QRS_NEXT_CUT()
PTP {E1 29337.004,E2 29337.004}
PTP {X 0,Y 607.899,A -85,B 0,C 180,E1 29337.004,E2 29337.004,E3 0,E4 0,E5 0,E6 0}
QRS_SPEED_INIT()
LIN {X 0,Y 607.899,Z 862.5,A -85,B 0,C 180,E1 29337.004,E2 29337.004,E3 0,E4 0,E5 0,E6 0} C_VEL
LIN {X 0,Y 607.899,Z 754.418,A -85,B 0,C 180,E1 29337.004,E2 29337.004} C_VEL
LIN {X 0,Y 607.899,Z 746.5,A -85,B 0,C 180,E1 29337.004,E2 29337.004} C_VEL
LIN {X 0,Y 607.901,Z 744.678,A -85,B 0,C 180,E1 29336.738,E2 29336.738} C_VEL
LIN {X 0,Y 607.905,Z 753.292,A -85,B 0,C 180,E1 29334.811,E2 29334.811} C_VEL
LIN {X 0,Y 607.912,Z 760.307,A -85,B 0,C 180,E1 29332.821,E2 29332.821} C_VEL
LIN {X 0,Y 607.912,Z 766.021,A -85,B 0,C 180,E1 29330.697,E2 29330.697} C_VEL
LIN {X 0,Y 607.897,Z 769.752,A -85,B 0,C 180,E1 29328.714,E2 29328.714} C_VEL
LIN {X 0,Y 607.897,Z 771.855,A -85,B 0,C 180,E1 29326.689,E2 29326.689} C_VEL
LIN {X 0,Y 607.9,Z 772.434,A -85,B 0,C 180,E1 29324.646,E2 29324.646} C_VEL
LIN {X 0,Y 607.91,Z 771.473,A -85,B 0,C 180,E1 29322.682,E2 29322.682} C_VEL
LIN {X 0,Y 607.91,Z 768.915,A -85,B 0,C 180,E1 29320.697,E2 29320.697} C_VEL
LIN {X 0,Y 607.9,Z 764.827,A -85,B 0,C 180,E1 29318.687,E2 29318.687} C_VEL
LIN {X 0,Y 607.898,Z 759.231,A -85,B 0,C 180,E1 29316.752,E2 29316.752} C_VEL
LIN {X 0,Y 607.902,Z 751.53,A -85,B 0,C 180,E1 29314.684,E2 29314.684} C_VEL
LIN {X 0,Y 607.918,Z 742.857,A -85,B 0,C 180,E1 29312.793,E2 29312.793} C_VEL
LIN {X 0,Y 607.917,Z 732.736,A -85,B 0,C 180,E1 29310.977,E2 29310.977} C_VEL
LIN {X 0,Y 607.91,Z 720.694,A -85,B 0,C 180,E1 29309.128,E2 29309.128} C_VEL
LIN {X 0,Y 607.913,Z 707.235,A -85,B 0,C 180,E1 29307.355,E2 29307.355} C_VEL
LIN {X 0,Y 607.916,Z 692.141,A -85,B 0,C 180,E1 29305.655,E2 29305.655} C_VEL
LIN {X 0,Y 607.915,Z 676.239,A -85,B 0,C 180,E1 29304.104,E2 29304.104} C_VEL
LIN {X 0,Y 607.912,Z 658.424,A -85,B 0,C 180,E1 29302.6,E2 29302.6} C_VEL
LIN {X 0,Y 607.917,Z 640.204,A -85,B 0,C 180,E1 29301.273,E2 29301.273} C_VEL
LIN {X 0,Y 607.917,Z 621.242,A -85,B 0,C 180,E1 29300.103,E2 29300.103} C_VEL
LIN {X 0,Y 607.914,Z 601.356,A -85,B 0,C 180,E1 29299.067,E2 29299.067} C_VEL
LIN {X 0,Y 607.915,Z 581.383,A -85,B 0,C 180,E1 29298.2,E2 29298.2} C_VEL
LIN {X 0,Y 607.915,Z 561.009,A -85,B 0,C 180,E1 29297.504,E2 29297.504} C_VEL
LIN {X 0,Y 607.899,Z 539.165,A -85,B 0,C 180,E1 29296.934,E2 29296.934} C_VEL
LIN {X 0,Y 607.904,Z 518.887,A -85,B 0,C 180,E1 29296.57,E2 29296.57} C_VEL
LIN {X 0,Y 607.912,Z 289.818,A -85,B 0,C 180,E1 29293.507,E2 29293.507} C_VEL
LIN {X 0,Y 607.887,Z 237.014,A -85,B 0,C 180,E1 29292.776,E2 29292.776} C_VEL
LIN {X 0,Y 607.91,Z 237.007,A -85,B 0,C 180,E1 29289.655,E2 29289.655} C_VEL
LIN {X 0,Y 607.874,Z 237.01,A -85,B 0,C 180,E1 29286.459,E2 29286.459} C_VEL
LIN {X 0,Y 607.915,Z 237.008,A -85,B 0,C 180,E1 29283.435,E2 29283.435} C_VEL
LIN {X 0,Y 607.87,Z 237.011,A -85,B 0,C 180,E1 29280.288,E2 29280.288} C_VEL
LIN {X 0,Y 607.913,Z 237.011,A -85,B 0,C 180,E1 29277.157,E2 29277.157} C_VEL
LIN {X 0,Y 607.868,Z 237.01,A -85,B 0,C 180,E1 29274.075,E2 29274.075} C_VEL
LIN {X 0,Y 607.917,Z 237.014,A -85,B 0,C 180,E1 29270.907,E2 29270.907} C_VEL
LIN {X 0,Y 607.874,Z 237.009,A -85,B 0,C 180,E1 29267.764,E2 29267.764} C_VEL
LIN {X 0,Y 607.886,Z 237.013,A -85,B 0,C 180,E1 29264.479,E2 29264.479} C_VEL
LIN {X 0,Y 607.895,Z 237.008,A -85,B 0,C 180,E1 29261.384,E2 29261.384} C_VEL
LIN {X 0,Y 607.872,Z 237.012,A -85,B 0,C 180,E1 29258.228,E2 29258.228} C_VEL
LIN {X 0,Y 607.903,Z 237.008,A -85,B 0,C 180,E1 29255.191,E2 29255.191} C_VEL
LIN {X 0,Y 607.863,Z 237.012,A -85,B 0,C 180,E1 29251.98,E2 29251.98} C_VEL
LIN {X 0,Y 607.917,Z 237.009,A -85,B 0,C 180,E1 29248.87,E2 29248.87} C_VEL
LIN {X 0,Y 607.858,Z 237.011,A -85,B 0,C 180,E1 29245.756,E2 29245.756} C_VEL
LIN {X 0,Y 607.916,Z 237.011,A -85,B 0,C 180,E1 29242.725,E2 29242.725} C_VEL
LIN {X 0,Y 607.856,Z 237.011,A -85,B 0,C 180,E1 29239.672,E2 29239.672} C_VEL
LIN {X 0,Y 607.917,Z 237.012,A -85,B 0,C 180,E1 29236.592,E2 29236.592} C_VEL
LIN {X 0,Y 607.854,Z 237.011,A -85,B 0,C 180,E1 29233.522,E2 29233.522} C_VEL
LIN {X 0,Y 607.918,Z 237.013,A -85,B 0,C 180,E1 29230.456,E2 29230.456} C_VEL
LIN {X 0,Y 607.851,Z 237.012,A -85,B 0,C 180,E1 29227.465,E2 29227.465} C_VEL
LIN {X 0,Y 607.918,Z 237.013,A -85,B 0,C 180,E1 29224.371,E2 29224.371} C_VEL
LIN {X 0,Y 607.849,Z 237.012,A -85,B 0,C 180,E1 29221.403,E2 29221.403} C_VEL
LIN {X 0,Y 607.916,Z 237.012,A -85,B 0,C 180,E1 29218.356,E2 29218.356} C_VEL
LIN {X 0,Y 607.846,Z 237.013,A -85,B 0,C 180,E1 29215.311,E2 29215.311} C_VEL
LIN {X 0,Y 607.919,Z 237.012,A -85,B 0,C 180,E1 29212.279,E2 29212.279} C_VEL
LIN {X 0,Y 607.844,Z 237.013,A -85,B 0,C 180,E1 29209.231,E2 29209.231} C_VEL
LIN {X 0,Y 607.919,Z 237.013,A -85,B 0,C 180,E1 29206.179,E2 29206.179} C_VEL
LIN {X 0,Y 607.84,Z 237.013,A -85,B 0,C 180,E1 29203.177,E2 29203.177} C_VEL
LIN {X 0,Y 607.912,Z 237.013,A -85,B 0,C 180,E1 29200.113,E2 29200.113} C_VEL
LIN {X 0,Y 607.839,Z 237.013,A -85,B 0,C 180,E1 29197.082,E2 29197.082} C_VEL
LIN {X 0,Y 607.915,Z 237.014,A -85,B 0,C 180,E1 29193.999,E2 29193.999} C_VEL
LIN {X 0,Y 607.836,Z 237.014,A -85,B 0,C 180,E1 29190.986,E2 29190.986} C_VEL
LIN {X 0,Y 607.915,Z 237.013,A -85,B 0,C 180,E1 29187.951,E2 29187.951} C_VEL
LIN {X 0,Y 607.834,Z 237.014,A -85,B 0,C 180,E1 29184.903,E2 29184.903} C_VEL
LIN {X 0,Y 607.904,Z 237.014,A -85,B 0,C 180,E1 29181.921,E2 29181.921} C_VEL
LIN {X 0,Y 607.833,Z 237.014,A -85,B 0,C 180,E1 29178.907,E2 29178.907} C_VEL
LIN {X 0,Y 607.888,Z 237.014,A -85,B 0,C 180,E1 29175.941,E2 29175.941} C_VEL
LIN {X 0,Y 607.833,Z 237.015,A -85,B 0,C 180,E1 29172.926,E2 29172.926} C_VEL
LIN {X 0,Y 607.844,Z 237.014,A -85,B 0,C 180,E1 29170.231,E2 29170.231} C_VEL
LIN {X 0,Y 607.839,Z 237.015,A -85,B 0,C 180,E1 29166.99,E2 29166.99} C_VEL
LIN {X 0,Y 607.835,Z 237.015,A -85,B 0,C 180,E1 29164.244,E2 29164.244} C_VEL
LIN {X 0,Y 607.843,Z 237.015,A -85,B 0,C 180,E1 29160.941,E2 29160.941} C_VEL
LIN {X 0,Y 607.834,Z 237.015,A -85,B 0,C 180,E1 29158.208,E2 29158.208} C_VEL
LIN {X 0,Y 607.858,Z 237.014,A -85,B 0,C 180,E1 29154.998,E2 29154.998} C_VEL
LIN {X 0,Y 607.836,Z 237.014,A -85,B 0,C 180,E1 29152.152,E2 29152.152} C_VEL
LIN {X 0,Y 607.871,Z 237.014,A -85,B 0,C 180,E1 29148.999,E2 29148.999} C_VEL
LIN {X 0,Y 607.834,Z 237.014,A -85,B 0,C 180,E1 29146.2,E2 29146.2} C_VEL
LIN {X 0,Y 607.894,Z 237.013,A -85,B 0,C 180,E1 29143.074,E2 29143.074} C_VEL
LIN {X 0,Y 607.835,Z 237.014,A -85,B 0,C 180,E1 29140.192,E2 29140.192} C_VEL
LIN {X 0,Y 607.915,Z 237.013,A -85,B 0,C 180,E1 29137.159,E2 29137.159} C_VEL
LIN {X 0,Y 607.837,Z 237.013,A -85,B 0,C 180,E1 29134.126,E2 29134.126} C_VEL
LIN {X 0,Y 607.914,Z 237.014,A -85,B 0,C 180,E1 29131.082,E2 29131.082} C_VEL
LIN {X 0,Y 607.84,Z 237.013,A -85,B 0,C 180,E1 29128.077,E2 29128.077} C_VEL
LIN {X 0,Y 607.918,Z 237.012,A -85,B 0,C 180,E1 29124.969,E2 29124.969} C_VEL
LIN {X 0,Y 607.843,Z 237.013,A -85,B 0,C 180,E1 29121.913,E2 29121.913} C_VEL
LIN {X 0,Y 607.918,Z 237.012,A -85,B 0,C 180,E1 29118.86,E2 29118.86} C_VEL
LIN {X 0,Y 607.845,Z 237.013,A -85,B 0,C 180,E1 29115.82,E2 29115.82} C_VEL
LIN {X 0,Y 607.918,Z 237.012,A -85,B 0,C 180,E1 29112.785,E2 29112.785} C_VEL
LIN {X 0,Y 607.848,Z 237.012,A -85,B 0,C 180,E1 29109.78,E2 29109.78} C_VEL
LIN {X 0,Y 607.919,Z 237.08,A -85,B 0,C 180,E1 29106.651,E2 29106.651} C_VEL
LIN {X 0,Y 607.92,Z 284.175,A -85,B 0,C 180,E1 29103.546,E2 29103.546} C_VEL
LIN {X 0,Y 607.916,Z 302.922,A -85,B 0,C 180,E1 29102.36,E2 29102.36} C_VEL
LIN {X 0,Y 607.905,Z 524.312,A -85,B 0,C 180,E1 29099.375,E2 29099.375} C_VEL
LIN {X 0,Y 607.903,Z 607.752,A -85,B 0,C 180,E1 29098.246,E2 29098.246} C_VEL
LIN {X 0,Y 607.908,Z 628.255,A -85,B 0,C 180,E1 29097.805,E2 29097.805} C_VEL
LIN {X 0,Y 607.907,Z 648.842,A -85,B 0,C 180,E1 29097.208,E2 29097.208} C_VEL
LIN {X 0,Y 607.913,Z 669.605,A -85,B 0,C 180,E1 29096.416,E2 29096.416} C_VEL
LIN {X 0,Y 607.918,Z 690.768,A -85,B 0,C 180,E1 29095.42,E2 29095.42} C_VEL
LIN {X 0,Y 607.916,Z 710.107,A -85,B 0,C 180,E1 29094.331,E2 29094.331} C_VEL
LIN {X 0,Y 607.914,Z 728.578,A -85,B 0,C 180,E1 29093.094,E2 29093.094} C_VEL
LIN {X 0,Y 607.911,Z 746.777,A -85,B 0,C 180,E1 29091.677,E2 29091.677} C_VEL
LIN {X 0,Y 607.913,Z 763.663,A -85,B 0,C 180,E1 29090.154,E2 29090.154} C_VEL
LIN {X 0,Y 607.918,Z 779.474,A -85,B 0,C 180,E1 29088.506,E2 29088.506} C_VEL
LIN {X 0,Y 607.913,Z 793.414,A -85,B 0,C 180,E1 29086.816,E2 29086.816} C_VEL
LIN {X 0,Y 607.918,Z 805.908,A -85,B 0,C 180,E1 29085.061,E2 29085.061} C_VEL
LIN {X 0,Y 607.919,Z 817.422,A -85,B 0,C 180,E1 29083.176,E2 29083.176} C_VEL
LIN {X 0,Y 607.912,Z 827.065,A -85,B 0,C 180,E1 29081.286,E2 29081.286} C_VEL
LIN {X 0,Y 607.911,Z 835.467,A -85,B 0,C 180,E1 29079.275,E2 29079.275} C_VEL
LIN {X 0,Y 607.91,Z 842.13,A -85,B 0,C 180,E1 29077.275,E2 29077.275} C_VEL
LIN {X 0,Y 607.914,Z 847.016,A -85,B 0,C 180,E1 29075.284,E2 29075.284} C_VEL
LIN {X 0,Y 607.917,Z 850.447,A -85,B 0,C 180,E1 29073.205,E2 29073.205} C_VEL
LIN {X 0,Y 607.91,Z 852.21,A -85,B 0,C 180,E1 29071.224,E2 29071.224} C_VEL
LIN {X 0,Y 607.902,Z 852.328,A -85,B 0,C 180,E1 29069.245,E2 29069.245} C_VEL
LIN {X 0,Y 607.908,Z 850.894,A -85,B 0,C 180,E1 29067.171,E2 29067.171} C_VEL
LIN {X 0,Y 607.912,Z 847.985,A -85,B 0,C 180,E1 29065.187,E2 29065.187} C_VEL
LIN {X 0,Y 607.915,Z 843.396,A -85,B 0,C 180,E1 29063.198,E2 29063.198} C_VEL
LIN {X 0,Y 607.906,Z 837.234,A -85,B 0,C 180,E1 29061.201,E2 29061.201} C_VEL
LIN {X 0,Y 607.899,Z 829.652,A -85,B 0,C 180,E1 29059.288,E2 29059.288} C_VEL
LIN {X 0,Y 607.899,Z 820.322,A -85,B 0,C 180,E1 29057.363,E2 29057.363} C_VEL
LIN {X 0,Y 607.904,Z 809.74,A -85,B 0,C 180,E1 29055.521,E2 29055.521} C_VEL
LIN {X 0,Y 607.911,Z 797.735,A -85,B 0,C 180,E1 29053.763,E2 29053.763} C_VEL
LIN {X 0,Y 607.906,Z 783.709,A -85,B 0,C 180,E1 29051.987,E2 29051.987} C_VEL
LIN {X 0,Y 607.908,Z 768.706,A -85,B 0,C 180,E1 29050.345,E2 29050.345} C_VEL
LIN {X 0,Y 607.916,Z 751.689,A -85,B 0,C 180,E1 29048.735,E2 29048.735} C_VEL
LIN {X 0,Y 607.918,Z 734.236,A -85,B 0,C 180,E1 29047.323,E2 29047.323} C_VEL
LIN {X 0,Y 607.915,Z 715.722,A -85,B 0,C 180,E1 29046.03,E2 29046.03} C_VEL
LIN {X 0,Y 607.918,Z 696.693,A -85,B 0,C 180,E1 29044.89,E2 29044.89} C_VEL
LIN {X 0,Y 607.9,Z 676.895,A -85,B 0,C 180,E1 29043.902,E2 29043.902} C_VEL
LIN {X 0,Y 607.907,Z 656.203,A -85,B 0,C 180,E1 29043.057,E2 29043.057} C_VEL
LIN {X 0,Y 607.918,Z 636.195,A -85,B 0,C 180,E1 29042.402,E2 29042.402} C_VEL
LIN {X 0,Y 607.904,Z 615.922,A -85,B 0,C 180,E1 29041.913,E2 29041.913} C_VEL
LIN {X 0,Y 607.914,Z 594.386,A -85,B 0,C 180,E1 29041.552,E2 29041.552} C_VEL
LIN {X 0,Y 607.881,Z 369.433,A -85,B 0,C 180,E1 29038.545,E2 29038.545} C_VEL
LIN {X 0,Y 607.916,Z 302.484,A -85,B 0,C 180,E1 29037.631,E2 29037.631} C_VEL
LIN {X 0,Y 607.865,Z 256.986,A -85,B 0,C 180,E1 29034.672,E2 29034.672} C_VEL
LIN {X 0,Y 607.919,Z 237.013,A -85,B 0,C 180,E1 29033.342,E2 29033.342} C_VEL
LIN {X 0,Y 607.846,Z 237.013,A -85,B 0,C 180,E1 29030.217,E2 29030.217} C_VEL
LIN {X 0,Y 607.919,Z 237.013,A -85,B 0,C 180,E1 29027.185,E2 29027.185} C_VEL
LIN {X 0,Y 607.843,Z 237.013,A -85,B 0,C 180,E1 29024.177,E2 29024.177} C_VEL
LIN {X 0,Y 607.919,Z 237.013,A -85,B 0,C 180,E1 29021.124,E2 29021.124} C_VEL
LIN {X 0,Y 607.838,Z 237.014,A -85,B 0,C 180,E1 29018.087,E2 29018.087} C_VEL
LIN {X 0,Y 607.919,Z 237.014,A -85,B 0,C 180,E1 29015.008,E2 29015.008} C_VEL
LIN {X 0,Y 607.834,Z 237.014,A -85,B 0,C 180,E1 29011.919,E2 29011.919} C_VEL
LIN {X 0,Y 607.906,Z 237.016,A -85,B 0,C 180,E1 29008.919,E2 29008.919} C_VEL
LIN {X 0,Y 607.829,Z 237.015,A -85,B 0,C 180,E1 29005.949,E2 29005.949} C_VEL
LIN {X 0,Y 607.892,Z 237.015,A -85,B 0,C 180,E1 29003.046,E2 29003.046} C_VEL
LIN {X 0,Y 607.829,Z 237.015,A -85,B 0,C 180,E1 29000.009,E2 29000.009} C_VEL
LIN {X 0,Y 607.869,Z 237.048,A -85,B 0,C 180,E1 28997.124,E2 28997.124} C_VEL
LIN {X 0,Y 607.9,Z 476.426,A -85,B 0,C 180,E1 28993.905,E2 28993.905} C_VEL
LIN {X 0,Y 607.902,Z 529.091,A -85,B 0,C 180,E1 28993.18,E2 28993.18} C_VEL
LIN {X 0,Y 607.918,Z 549.308,A -85,B 0,C 180,E1 28992.733,E2 28992.733} C_VEL
LIN {X 0,Y 607.901,Z 570.449,A -85,B 0,C 180,E1 28992.106,E2 28992.106} C_VEL
LIN {X 0,Y 607.901,Z 590.463,A -85,B 0,C 180,E1 28991.336,E2 28991.336} C_VEL
LIN {X 0,Y 607.919,Z 610.908,A -85,B 0,C 180,E1 28990.368,E2 28990.368} C_VEL
LIN {X 0,Y 607.917,Z 630.263,A -85,B 0,C 180,E1 28989.277,E2 28989.277} C_VEL
LIN {X 0,Y 607.914,Z 648.753,A -85,B 0,C 180,E1 28988.038,E2 28988.038} C_VEL
LIN {X 0,Y 607.913,Z 667.016,A -85,B 0,C 180,E1 28986.612,E2 28986.612} C_VEL
LIN {X 0,Y 607.915,Z 683.795,A -85,B 0,C 180,E1 28985.097,E2 28985.097} C_VEL
LIN {X 0,Y 607.915,Z 699.232,A -85,B 0,C 180,E1 28983.49,E2 28983.49} C_VEL
LIN {X 0,Y 607.916,Z 713.253,A -85,B 0,C 180,E1 28981.792,E2 28981.792} C_VEL
LIN {X 0,Y 607.914,Z 726.007,A -85,B 0,C 180,E1 28980.001,E2 28980.001} C_VEL
LIN {X 0,Y 607.913,Z 737.503,A -85,B 0,C 180,E1 28978.116,E2 28978.116} C_VEL
LIN {X 0,Y 607.901,Z 744.678,A -85,B 0,C 180,E1 28976.738,E2 28976.738} C_VEL
LIN {X 0,Y 606.904,Z 747.955,A -85,B 0,C 180,E1 28976.076,E2 28976.076} C_VEL
LIN {X 0,Y 600.672,Z 755.675,A -85,B 0,C 180,E1 28974.293,E2 28974.293} C_VEL
LIN {X 0,Y 599.922,Z 757.876,A -85,B 0,C 180,E1 28973.696,E2 28973.696} C_VEL
LIN {X 0,Y 599.92,Z 763.885,A -85,B 0,C 180,E1 28971.664,E2 28971.664} C_VEL
LIN {X 0,Y 599.91,Z 768.491,A -85,B 0,C 180,E1 28969.528,E2 28969.528} C_VEL
LIN {X 0,Y 599.902,Z 771.287,A -85,B 0,C 180,E1 28967.488,E2 28967.488} C_VEL
LIN {X 0,Y 599.91,Z 772.4,A -85,B 0,C 180,E1 28965.425,E2 28965.425} C_VEL
LIN {X 0,Y 599.917,Z 771.889,A -85,B 0,C 180,E1 28963.244,E2 28963.244} C_VEL
LIN {X 0,Y 599.915,Z 769.843,A -85,B 0,C 180,E1 28961.204,E2 28961.204} C_VEL
LIN {X 0,Y 599.918,Z 766.178,A -85,B 0,C 180,E1 28959.209,E2 28959.209} C_VEL
LIN {X 0,Y 599.921,Z 760.511,A -85,B 0,C 180,E1 28957.048,E2 28957.048} C_VEL
LIN {X 0,Y 599.933,Z 753.6,A -85,B 0,C 180,E1 28955.046,E2 28955.046} C_VEL
LIN {X 0,Y 599.947,Z 744.835,A -85,B 0,C 180,E1 28953.046,E2 28953.046} C_VEL
LIN {X 0,Y 599.973,Z 733.944,A -85,B 0,C 180,E1 28950.993,E2 28950.993} C_VEL
LIN {X 0,Y 600.007,Z 722.136,A -85,B 0,C 180,E1 28949.116,E2 28949.116} C_VEL
LIN {X 0,Y 600.052,Z 708.647,A -85,B 0,C 180,E1 28947.297,E2 28947.297} C_VEL
LIN {X 0,Y 600.123,Z 693.662,A -85,B 0,C 180,E1 28945.56,E2 28945.56} C_VEL
LIN {X 0,Y 600.203,Z 677.026,A -85,B 0,C 180,E1 28943.896,E2 28943.896} C_VEL
LIN {X 0,Y 600.292,Z 660.221,A -85,B 0,C 180,E1 28942.441,E2 28942.441} C_VEL
LIN {X 0,Y 600.386,Z 641.597,A -85,B 0,C 180,E1 28941.053,E2 28941.053} C_VEL
LIN {X 0,Y 600.481,Z 622.419,A -85,B 0,C 180,E1 28939.843,E2 28939.843} C_VEL
LIN {X 0,Y 600.59,Z 601.315,A -85,B 0,C 180,E1 28938.725,E2 28938.725} C_VEL
LIN {X 0,Y 600.687,Z 580.897,A -85,B 0,C 180,E1 28937.833,E2 28937.833} C_VEL
LIN {X 0,Y 600.755,Z 559.86,A -85,B 0,C 180,E1 28937.113,E2 28937.113} C_VEL
LIN {X 0,Y 600.816,Z 537.813,A -85,B 0,C 180,E1 28936.545,E2 28936.545} C_VEL
LIN {X 0,Y 600.867,Z 516.414,A -85,B 0,C 180,E1 28936.169,E2 28936.169} C_VEL
LIN {X 0,Y 601.082,Z 290.741,A -85,B 0,C 180,E1 28933.121,E2 28933.121} C_VEL
LIN {X 0,Y 600.973,Z 241.06,A -85,B 0,C 180,E1 28932.427,E2 28932.427} C_VEL
LIN {X 0,Y 599.935,Z 238.001,A -85,B 0,C 180,E1 28932.299,E2 28932.299} C_VEL
LIN {X 0,Y 599.976,Z 238.003,A -85,B 0,C 180,E1 28929.169,E2 28929.169} C_VEL
LIN {X 0,Y 599.941,Z 237.996,A -85,B 0,C 180,E1 28926.038,E2 28926.038} C_VEL
LIN {X 0,Y 599.959,Z 238.003,A -85,B 0,C 180,E1 28922.795,E2 28922.795} C_VEL
LIN {X 0,Y 599.973,Z 237.995,A -85,B 0,C 180,E1 28919.556,E2 28919.556} C_VEL
LIN {X 0,Y 599.932,Z 238.001,A -85,B 0,C 180,E1 28916.317,E2 28916.317} C_VEL
LIN {X 0,Y 599.977,Z 237.997,A -85,B 0,C 180,E1 28913.264,E2 28913.264} C_VEL
LIN {X 0,Y 599.93,Z 238,A -85,B 0,C 180,E1 28910.182,E2 28910.182} C_VEL
LIN {X 0,Y 599.975,Z 237.999,A -85,B 0,C 180,E1 28907.057,E2 28907.057} C_VEL
LIN {X 0,Y 599.926,Z 237.999,A -85,B 0,C 180,E1 28903.985,E2 28903.985} C_VEL
LIN {X 0,Y 599.976,Z 238.002,A -85,B 0,C 180,E1 28900.855,E2 28900.855} C_VEL
LIN {X 0,Y 599.925,Z 237.999,A -85,B 0,C 180,E1 28897.759,E2 28897.759} C_VEL
LIN {X 0,Y 599.973,Z 238.003,A -85,B 0,C 180,E1 28894.589,E2 28894.589} C_VEL
LIN {X 0,Y 599.929,Z 237.998,A -85,B 0,C 180,E1 28891.529,E2 28891.529} C_VEL
LIN {X 0,Y 599.945,Z 238.002,A -85,B 0,C 180,E1 28888.282,E2 28888.282} C_VEL
LIN {X 0,Y 599.943,Z 237.997,A -85,B 0,C 180,E1 28885.221,E2 28885.221} C_VEL
LIN {X 0,Y 599.925,Z 238.001,A -85,B 0,C 180,E1 28881.953,E2 28881.953} C_VEL
LIN {X 0,Y 599.969,Z 237.998,A -85,B 0,C 180,E1 28878.855,E2 28878.855} C_VEL
LIN {X 0,Y 599.917,Z 238.001,A -85,B 0,C 180,E1 28875.721,E2 28875.721} C_VEL
LIN {X 0,Y 599.975,Z 237.999,A -85,B 0,C 180,E1 28872.645,E2 28872.645} C_VEL
LIN {X 0,Y 599.913,Z 238.001,A -85,B 0,C 180,E1 28869.514,E2 28869.514} C_VEL
LIN {X 0,Y 599.979,Z 238.001,A -85,B 0,C 180,E1 28866.423,E2 28866.423} C_VEL
LIN {X 0,Y 599.911,Z 238.001,A -85,B 0,C 180,E1 28863.364,E2 28863.364} C_VEL
LIN {X 0,Y 599.978,Z 238.004,A -85,B 0,C 180,E1 28860.225,E2 28860.225} C_VEL
LIN {X 0,Y 599.912,Z 238,A -85,B 0,C 180,E1 28857.136,E2 28857.136} C_VEL
LIN {X 0,Y 599.946,Z 238.003,A -85,B 0,C 180,E1 28853.925,E2 28853.925} C_VEL
LIN {X 0,Y 599.909,Z 238.001,A -85,B 0,C 180,E1 28851.074,E2 28851.074} C_VEL
LIN {X 0,Y 599.947,Z 238.004,A -85,B 0,C 180,E1 28847.867,E2 28847.867} C_VEL
LIN {X 0,Y 599.907,Z 238.001,A -85,B 0,C 180,E1 28844.962,E2 28844.962} C_VEL
LIN {X 0,Y 599.948,Z 238.004,A -85,B 0,C 180,E1 28841.805,E2 28841.805} C_VEL
LIN {X 0,Y 599.904,Z 238.002,A -85,B 0,C 180,E1 28838.893,E2 28838.893} C_VEL
LIN {X 0,Y 599.949,Z 238.003,A -85,B 0,C 180,E1 28835.748,E2 28835.748} C_VEL
LIN {X 0,Y 599.901,Z 238.002,A -85,B 0,C 180,E1 28832.796,E2 28832.796} C_VEL
LIN {X 0,Y 599.947,Z 238.004,A -85,B 0,C 180,E1 28829.666,E2 28829.666} C_VEL
LIN {X 0,Y 599.898,Z 238.002,A -85,B 0,C 180,E1 28826.742,E2 28826.742} C_VEL
LIN {X 0,Y 599.959,Z 238.004,A -85,B 0,C 180,E1 28823.679,E2 28823.679} C_VEL
LIN {X 0,Y 599.894,Z 238.003,A -85,B 0,C 180,E1 28820.69,E2 28820.69} C_VEL
LIN {X 0,Y 599.957,Z 238.004,A -85,B 0,C 180,E1 28817.591,E2 28817.591} C_VEL
LIN {X 0,Y 599.891,Z 238.003,A -85,B 0,C 180,E1 28814.674,E2 28814.674} C_VEL
LIN {X 0,Y 599.972,Z 238.004,A -85,B 0,C 180,E1 28811.632,E2 28811.632} C_VEL
LIN {X 0,Y 599.889,Z 238.004,A -85,B 0,C 180,E1 28808.626,E2 28808.626} C_VEL
LIN {X 0,Y 599.967,Z 238.004,A -85,B 0,C 180,E1 28805.641,E2 28805.641} C_VEL
LIN {X 0,Y 599.886,Z 238.004,A -85,B 0,C 180,E1 28802.578,E2 28802.578} C_VEL
LIN {X 0,Y 599.961,Z 238.004,A -85,B 0,C 180,E1 28799.617,E2 28799.617} C_VEL
LIN {X 0,Y 599.891,Z 238.004,A -85,B 0,C 180,E1 28796.559,E2 28796.559} C_VEL
LIN {X 0,Y 599.956,Z 238.003,A -85,B 0,C 180,E1 28793.588,E2 28793.588} C_VEL
LIN {X 0,Y 599.893,Z 238.003,A -85,B 0,C 180,E1 28790.501,E2 28790.501} C_VEL
LIN {X 0,Y 599.947,Z 238.004,A -85,B 0,C 180,E1 28787.577,E2 28787.577} C_VEL
LIN {X 0,Y 599.897,Z 238.003,A -85,B 0,C 180,E1 28784.433,E2 28784.433} C_VEL
LIN {X 0,Y 599.948,Z 238.004,A -85,B 0,C 180,E1 28781.487,E2 28781.487} C_VEL
LIN {X 0,Y 599.9,Z 238.002,A -85,B 0,C 180,E1 28778.386,E2 28778.386} C_VEL
LIN {X 0,Y 599.942,Z 238.003,A -85,B 0,C 180,E1 28775.481,E2 28775.481} C_VEL
LIN {X 0,Y 599.907,Z 238.002,A -85,B 0,C 180,E1 28772.396,E2 28772.396} C_VEL
LIN {X 0,Y 599.931,Z 238.003,A -85,B 0,C 180,E1 28769.498,E2 28769.498} C_VEL
LIN {X 0,Y 599.908,Z 238.002,A -85,B 0,C 180,E1 28766.268,E2 28766.268} C_VEL
LIN {X 0,Y 599.939,Z 238.004,A -85,B 0,C 180,E1 28763.37,E2 28763.37} C_VEL
LIN {X 0,Y 599.911,Z 238.002,A -85,B 0,C 180,E1 28760.202,E2 28760.202} C_VEL
LIN {X 0,Y 599.941,Z 238.004,A -85,B 0,C 180,E1 28757.288,E2 28757.288} C_VEL
LIN {X 0,Y 599.912,Z 238.002,A -85,B 0,C 180,E1 28754.082,E2 28754.082} C_VEL
LIN {X 0,Y 599.965,Z 238.004,A -85,B 0,C 180,E1 28751.04,E2 28751.04} C_VEL
LIN {X 0,Y 599.913,Z 238.003,A -85,B 0,C 180,E1 28747.95,E2 28747.95} C_VEL
LIN {X 0,Y 599.978,Z 238.232,A -85,B 0,C 180,E1 28747.139,E2 28747.139} C_VEL
LIN {X 0,Y 601.065,Z 241.208,A -85,B 0,C 180,E1 28746.857,E2 28746.857} C_VEL
LIN {X 0,Y 600.904,Z 286.795,A -85,B 0,C 180,E1 28743.818,E2 28743.818} C_VEL
LIN {X 0,Y 600.96,Z 303.158,A -85,B 0,C 180,E1 28742.778,E2 28742.778} C_VEL
LIN {X 0,Y 600.982,Z 464.512,A -85,B 0,C 180,E1 28740.557,E2 28740.557} C_VEL
LIN {X 0,Y 600.847,Z 607.966,A -85,B 0,C 180,E1 28738.605,E2 28738.605} C_VEL
LIN {X 0,Y 600.789,Z 628.958,A -85,B 0,C 180,E1 28738.145,E2 28738.145} C_VEL
LIN {X 0,Y 600.712,Z 649.582,A -85,B 0,C 180,E1 28737.534,E2 28737.534} C_VEL
LIN {X 0,Y 600.646,Z 669.608,A -85,B 0,C 180,E1 28736.761,E2 28736.761} C_VEL
LIN {X 0,Y 600.54,Z 690.771,A -85,B 0,C 180,E1 28735.755,E2 28735.755} C_VEL
LIN {X 0,Y 600.445,Z 710.128,A -85,B 0,C 180,E1 28734.652,E2 28734.652} C_VEL
LIN {X 0,Y 600.355,Z 728.425,A -85,B 0,C 180,E1 28733.414,E2 28733.414} C_VEL
LIN {X 0,Y 600.25,Z 746.287,A -85,B 0,C 180,E1 28732.01,E2 28732.01} C_VEL
LIN {X 0,Y 600.165,Z 763.156,A -85,B 0,C 180,E1 28730.477,E2 28730.477} C_VEL
LIN {X 0,Y 600.102,Z 778.669,A -85,B 0,C 180,E1 28728.85,E2 28728.85} C_VEL
LIN {X 0,Y 600.048,Z 792.568,A -85,B 0,C 180,E1 28727.152,E2 28727.152} C_VEL
LIN {X 0,Y 599.999,Z 805.91,A -85,B 0,C 180,E1 28725.265,E2 28725.265} C_VEL
LIN {X 0,Y 599.958,Z 817.217,A -85,B 0,C 180,E1 28723.393,E2 28723.393} C_VEL
LIN {X 0,Y 599.931,Z 826.837,A -85,B 0,C 180,E1 28721.486,E2 28721.486} C_VEL
LIN {X 0,Y 599.915,Z 835.113,A -85,B 0,C 180,E1 28719.496,E2 28719.496} C_VEL
LIN {X 0,Y 599.912,Z 841.875,A -85,B 0,C 180,E1 28717.469,E2 28717.469} C_VEL
LIN {X 0,Y 599.915,Z 846.811,A -85,B 0,C 180,E1 28715.45,E2 28715.45} C_VEL
LIN {X 0,Y 599.916,Z 850.37,A -85,B 0,C 180,E1 28713.313,E2 28713.313} C_VEL
LIN {X 0,Y 599.909,Z 852.21,A -85,B 0,C 180,E1 28711.241,E2 28711.241} C_VEL
LIN {X 0,Y 599.902,Z 852.328,A -85,B 0,C 180,E1 28709.235,E2 28709.235} C_VEL
LIN {X 0,Y 599.909,Z 850.894,A -85,B 0,C 180,E1 28707.133,E2 28707.133} C_VEL
LIN {X 0,Y 599.914,Z 847.985,A -85,B 0,C 180,E1 28705.123,E2 28705.123} C_VEL
LIN {X 0,Y 599.92,Z 843.396,A -85,B 0,C 180,E1 28703.107,E2 28703.107} C_VEL
LIN {X 0,Y 599.924,Z 837.235,A -85,B 0,C 180,E1 28701.083,E2 28701.083} C_VEL
LIN {X 0,Y 599.923,Z 829.653,A -85,B 0,C 180,E1 28699.144,E2 28699.144} C_VEL
LIN {X 0,Y 599.942,Z 820.093,A -85,B 0,C 180,E1 28697.15,E2 28697.15} C_VEL
LIN {X 0,Y 599.978,Z 809.104,A -85,B 0,C 180,E1 28695.227,E2 28695.227} C_VEL
LIN {X 0,Y 600.013,Z 797.029,A -85,B 0,C 180,E1 28693.443,E2 28693.443} C_VEL
LIN {X 0,Y 600.082,Z 782.859,A -85,B 0,C 180,E1 28691.644,E2 28691.644} C_VEL
LIN {X 0,Y 600.156,Z 767.187,A -85,B 0,C 180,E1 28689.928,E2 28689.928} C_VEL
LIN {X 0,Y 600.243,Z 750.582,A -85,B 0,C 180,E1 28688.356,E2 28688.356} C_VEL
LIN {X 0,Y 600.318,Z 732.788,A -85,B 0,C 180,E1 28686.906,E2 28686.906} C_VEL
LIN {X 0,Y 600.421,Z 714.12,A -85,B 0,C 180,E1 28685.607,E2 28685.607} C_VEL
LIN {X 0,Y 600.533,Z 693.714,A -85,B 0,C 180,E1 28684.401,E2 28684.401} C_VEL
LIN {X 0,Y 600.607,Z 674.531,A -85,B 0,C 180,E1 28683.449,E2 28683.449} C_VEL
LIN {X 0,Y 600.695,Z 653.94,A -85,B 0,C 180,E1 28682.624,E2 28682.624} C_VEL
LIN {X 0,Y 600.79,Z 632.305,A -85,B 0,C 180,E1 28681.942,E2 28681.942} C_VEL
LIN {X 0,Y 600.828,Z 612.544,A -85,B 0,C 180,E1 28681.482,E2 28681.482} C_VEL
LIN {X 0,Y 600.891,Z 583.533,A -85,B 0,C 180,E1 28681.043,E2 28681.043} C_VEL
LIN {X 0,Y 601.06,Z 360.357,A -85,B 0,C 180,E1 28678.021,E2 28678.021} C_VEL
LIN {X 0,Y 600.94,Z 303.057,A -85,B 0,C 180,E1 28677.22,E2 28677.22} C_VEL
LIN {X 0,Y 600.956,Z 260.62,A -85,B 0,C 180,E1 28674.448,E2 28674.448} C_VEL
LIN {X 0,Y 601.064,Z 241.21,A -85,B 0,C 180,E1 28673.143,E2 28673.143} C_VEL
LIN {X 0,Y 599.94,Z 238.006,A -85,B 0,C 180,E1 28672.81,E2 28672.81} C_VEL
LIN {X 0,Y 599.916,Z 238.002,A -85,B 0,C 180,E1 28669.907,E2 28669.907} C_VEL
LIN {X 0,Y 599.924,Z 238.004,A -85,B 0,C 180,E1 28666.607,E2 28666.607} C_VEL
LIN {X 0,Y 599.917,Z 238.002,A -85,B 0,C 180,E1 28663.762,E2 28663.762} C_VEL
LIN {X 0,Y 599.911,Z 238.003,A -85,B 0,C 180,E1 28660.417,E2 28660.417} C_VEL
LIN {X 0,Y 599.92,Z 238.002,A -85,B 0,C 180,E1 28657.59,E2 28657.59} C_VEL
LIN {X 0,Y 599.912,Z 238.004,A -85,B 0,C 180,E1 28654.403,E2 28654.403} C_VEL
LIN {X 0,Y 599.912,Z 238.003,A -85,B 0,C 180,E1 28651.557,E2 28651.557} C_VEL
LIN {X 0,Y 599.902,Z 238.004,A -85,B 0,C 180,E1 28648.252,E2 28648.252} C_VEL
LIN {X 0,Y 599.907,Z 238.004,A -85,B 0,C 180,E1 28645.469,E2 28645.469} C_VEL
LIN {X 0,Y 599.901,Z 238.005,A -85,B 0,C 180,E1 28642.232,E2 28642.232} C_VEL
LIN {X 0,Y 599.898,Z 238.005,A -85,B 0,C 180,E1 28639.473,E2 28639.473} C_VEL
LIN {X 0,Y 599.912,Z 238.159,A -85,B 0,C 180,E1 28637.588,E2 28637.588} C_VEL
LIN {X 0,Y 601.095,Z 242.026,A -85,B 0,C 180,E1 28637.462,E2 28637.462} C_VEL
LIN {X 0,Y 600.895,Z 479.792,A -85,B 0,C 180,E1 28634.23,E2 28634.23} C_VEL
LIN {X 0,Y 600.837,Z 529.695,A -85,B 0,C 180,E1 28633.531,E2 28633.531} C_VEL
LIN {X 0,Y 600.797,Z 550.734,A -85,B 0,C 180,E1 28633.055,E2 28633.055} C_VEL
LIN {X 0,Y 600.694,Z 572.744,A -85,B 0,C 180,E1 28632.376,E2 28632.376} C_VEL
LIN {X 0,Y 600.619,Z 593.04,A -85,B 0,C 180,E1 28631.573,E2 28631.573} C_VEL
LIN {X 0,Y 600.537,Z 612.809,A -85,B 0,C 180,E1 28630.602,E2 28630.602} C_VEL
LIN {X 0,Y 600.426,Z 632.69,A -85,B 0,C 180,E1 28629.442,E2 28629.442} C_VEL
LIN {X 0,Y 600.336,Z 651.613,A -85,B 0,C 180,E1 28628.14,E2 28628.14} C_VEL
LIN {X 0,Y 600.245,Z 669.44,A -85,B 0,C 180,E1 28626.697,E2 28626.697} C_VEL
LIN {X 0,Y 600.16,Z 685.844,A -85,B 0,C 180,E1 28625.163,E2 28625.163} C_VEL
LIN {X 0,Y 600.082,Z 701.775,A -85,B 0,C 180,E1 28623.44,E2 28623.44} C_VEL
LIN {X 0,Y 600.039,Z 715.549,A -85,B 0,C 180,E1 28621.72,E2 28621.72} C_VEL
LIN {X 0,Y 599.991,Z 728.568,A -85,B 0,C 180,E1 28619.81,E2 28619.81} C_VEL
LIN {X 0,Y 599.953,Z 739.592,A -85,B 0,C 180,E1 28617.9,E2 28617.9} C_VEL
LIN {X 0,Y 599.936,Z 748.915,A -85,B 0,C 180,E1 28615.988,E2 28615.988} C_VEL
LIN {X 0,Y 599.918,Z 756.513,A -85,B 0,C 180,E1 28614.07,E2 28614.07} C_VEL
LIN {X 0,Y 599.922,Z 757.876,A -85,B 0,C 180,E1 28613.696,E2 28613.696} C_VEL
LIN {X 0,Y 598.927,Z 760.234,A -85,B 0,C 180,E1 28612.995,E2 28612.995} C_VEL
LIN {X 0,Y 592.561,Z 765.599,A -85,B 0,C 180,E1 28611.051,E2 28611.051} C_VEL
LIN {X 0,Y 591.917,Z 766.826,A -85,B 0,C 180,E1 28610.474,E2 28610.474} C_VEL
LIN {X 0,Y 591.914,Z 770.382,A -85,B 0,C 180,E1 28608.307,E2 28608.307} C_VEL
LIN {X 0,Y 591.914,Z 772.202,A -85,B 0,C 180,E1 28606.223,E2 28606.223} C_VEL
LIN {X 0,Y 591.91,Z 772.32,A -85,B 0,C 180,E1 28604.12,E2 28604.12} C_VEL
LIN {X 0,Y 591.905,Z 770.836,A -85,B 0,C 180,E1 28601.995,E2 28601.995} C_VEL
LIN {X 0,Y 591.905,Z 767.829,A -85,B 0,C 180,E1 28599.919,E2 28599.919} C_VEL
LIN {X 0,Y 591.91,Z 763.155,A -85,B 0,C 180,E1 28597.873,E2 28597.873} C_VEL
LIN {X 0,Y 591.93,Z 756.706,A -85,B 0,C 180,E1 28595.768,E2 28595.768} C_VEL
LIN {X 0,Y 591.962,Z 748.838,A -85,B 0,C 180,E1 28593.753,E2 28593.753} C_VEL
LIN {X 0,Y 592.001,Z 739.315,A -85,B 0,C 180,E1 28591.779,E2 28591.779} C_VEL
LIN {X 0,Y 592.076,Z 727.876,A -85,B 0,C 180,E1 28589.788,E2 28589.788} C_VEL
LIN {X 0,Y 592.169,Z 715.498,A -85,B 0,C 180,E1 28587.953,E2 28587.953} C_VEL
LIN {X 0,Y 592.267,Z 701.193,A -85,B 0,C 180,E1 28586.147,E2 28586.147} C_VEL
LIN {X 0,Y 592.41,Z 685.551,A -85,B 0,C 180,E1 28584.441,E2 28584.441} C_VEL
LIN {X 0,Y 592.593,Z 667.936,A -85,B 0,C 180,E1 28582.787,E2 28582.787} C_VEL
LIN {X 0,Y 592.798,Z 650.117,A -85,B 0,C 180,E1 28581.346,E2 28581.346} C_VEL
LIN {X 0,Y 592.985,Z 631.034,A -85,B 0,C 180,E1 28580.03,E2 28580.03} C_VEL
LIN {X 0,Y 593.182,Z 611.434,A -85,B 0,C 180,E1 28578.891,E2 28578.891} C_VEL
LIN {X 0,Y 593.392,Z 590.744,A -85,B 0,C 180,E1 28577.888,E2 28577.888} C_VEL
LIN {X 0,Y 593.553,Z 570.26,A -85,B 0,C 180,E1 28577.084,E2 28577.084} C_VEL
LIN {X 0,Y 593.695,Z 548.833,A -85,B 0,C 180,E1 28576.438,E2 28576.438} C_VEL
LIN {X 0,Y 593.818,Z 526.923,A -85,B 0,C 180,E1 28575.961,E2 28575.961} C_VEL
LIN {X 0,Y 594.281,Z 291.09,A -85,B 0,C 180,E1 28572.717,E2 28572.717} C_VEL
LIN {X 0,Y 594.203,Z 243.574,A -85,B 0,C 180,E1 28572.045,E2 28572.045} C_VEL
LIN {X 0,Y 592.331,Z 240.416,A -85,B 0,C 180,E1 28571.883,E2 28571.883} C_VEL
LIN {X 0,Y 592.024,Z 238.988,A -85,B 0,C 180,E1 28571.823,E2 28571.823} C_VEL
LIN {X 0,Y 591.999,Z 238.985,A -85,B 0,C 180,E1 28568.553,E2 28568.553} C_VEL
LIN {X 0,Y 592.035,Z 238.984,A -85,B 0,C 180,E1 28565.4,E2 28565.4} C_VEL
LIN {X 0,Y 591.994,Z 238.989,A -85,B 0,C 180,E1 28562.257,E2 28562.257} C_VEL
LIN {X 0,Y 592.036,Z 238.991,A -85,B 0,C 180,E1 28559.104,E2 28559.104} C_VEL
LIN {X 0,Y 591.996,Z 238.987,A -85,B 0,C 180,E1 28555.941,E2 28555.941} C_VEL
LIN {X 0,Y 592.017,Z 238.992,A -85,B 0,C 180,E1 28552.649,E2 28552.649} C_VEL
LIN {X 0,Y 592.028,Z 238.985,A -85,B 0,C 180,E1 28549.434,E2 28549.434} C_VEL
LIN {X 0,Y 591.991,Z 238.989,A -85,B 0,C 180,E1 28546.182,E2 28546.182} C_VEL
LIN {X 0,Y 592.039,Z 238.986,A -85,B 0,C 180,E1 28543.08,E2 28543.08} C_VEL
LIN {X 0,Y 591.986,Z 238.989,A -85,B 0,C 180,E1 28539.921,E2 28539.921} C_VEL
LIN {X 0,Y 592.039,Z 238.992,A -85,B 0,C 180,E1 28536.693,E2 28536.693} C_VEL
LIN {X 0,Y 591.995,Z 238.987,A -85,B 0,C 180,E1 28533.505,E2 28533.505} C_VEL
LIN {X 0,Y 591.997,Z 238.99,A -85,B 0,C 180,E1 28530.194,E2 28530.194} C_VEL
LIN {X 0,Y 592.022,Z 238.986,A -85,B 0,C 180,E1 28527.097,E2 28527.097} C_VEL
LIN {X 0,Y 591.983,Z 238.99,A -85,B 0,C 180,E1 28523.893,E2 28523.893} C_VEL
LIN {X 0,Y 592.041,Z 238.986,A -85,B 0,C 180,E1 28520.769,E2 28520.769} C_VEL
LIN {X 0,Y 591.979,Z 238.989,A -85,B 0,C 180,E1 28517.615,E2 28517.615} C_VEL
LIN {X 0,Y 592.039,Z 238.99,A -85,B 0,C 180,E1 28514.525,E2 28514.525} C_VEL
LIN {X 0,Y 591.977,Z 238.989,A -85,B 0,C 180,E1 28511.385,E2 28511.385} C_VEL
LIN {X 0,Y 592.021,Z 238.992,A -85,B 0,C 180,E1 28508.19,E2 28508.19} C_VEL
LIN {X 0,Y 591.983,Z 238.989,A -85,B 0,C 180,E1 28505.131,E2 28505.131} C_VEL
LIN {X 0,Y 591.986,Z 238.991,A -85,B 0,C 180,E1 28501.778,E2 28501.778} C_VEL
LIN {X 0,Y 591.991,Z 238.989,A -85,B 0,C 180,E1 28498.882,E2 28498.882} C_VEL
LIN {X 0,Y 591.982,Z 238.992,A -85,B 0,C 180,E1 28495.66,E2 28495.66} C_VEL
LIN {X 0,Y 591.998,Z 238.988,A -85,B 0,C 180,E1 28492.698,E2 28492.698} C_VEL
LIN {X 0,Y 591.971,Z 238.991,A -85,B 0,C 180,E1 28489.439,E2 28489.439} C_VEL
LIN {X 0,Y 592.017,Z 238.989,A -85,B 0,C 180,E1 28486.427,E2 28486.427} C_VEL
LIN {X 0,Y 591.965,Z 238.991,A -85,B 0,C 180,E1 28483.285,E2 28483.285} C_VEL
LIN {X 0,Y 592.024,Z 238.99,A -85,B 0,C 180,E1 28480.24,E2 28480.24} C_VEL
LIN {X 0,Y 591.963,Z 238.992,A -85,B 0,C 180,E1 28477.136,E2 28477.136} C_VEL
LIN {X 0,Y 592.033,Z 238.989,A -85,B 0,C 180,E1 28474.102,E2 28474.102} C_VEL
LIN {X 0,Y 591.959,Z 238.991,A -85,B 0,C 180,E1 28471.006,E2 28471.006} C_VEL
LIN {X 0,Y 592.035,Z 238.993,A -85,B 0,C 180,E1 28467.89,E2 28467.89} C_VEL
LIN {X 0,Y 591.956,Z 238.991,A -85,B 0,C 180,E1 28464.869,E2 28464.869} C_VEL
LIN {X 0,Y 592.037,Z 238.993,A -85,B 0,C 180,E1 28461.809,E2 28461.809} C_VEL
LIN {X 0,Y 591.954,Z 238.992,A -85,B 0,C 180,E1 28458.717,E2 28458.717} C_VEL
LIN {X 0,Y 592.018,Z 238.993,A -85,B 0,C 180,E1 28455.575,E2 28455.575} C_VEL
LIN {X 0,Y 591.951,Z 238.993,A -85,B 0,C 180,E1 28452.584,E2 28452.584} C_VEL
LIN {X 0,Y 592.018,Z 238.993,A -85,B 0,C 180,E1 28449.499,E2 28449.499} C_VEL
LIN {X 0,Y 591.949,Z 238.993,A -85,B 0,C 180,E1 28446.594,E2 28446.594} C_VEL
LIN {X 0,Y 592.023,Z 238.994,A -85,B 0,C 180,E1 28443.484,E2 28443.484} C_VEL
LIN {X 0,Y 591.949,Z 238.992,A -85,B 0,C 180,E1 28440.483,E2 28440.483} C_VEL
LIN {X 0,Y 592.027,Z 238.992,A -85,B 0,C 180,E1 28437.385,E2 28437.385} C_VEL
LIN {X 0,Y 591.952,Z 238.992,A -85,B 0,C 180,E1 28434.377,E2 28434.377} C_VEL
LIN {X 0,Y 592.022,Z 238.992,A -85,B 0,C 180,E1 28431.256,E2 28431.256} C_VEL
LIN {X 0,Y 591.954,Z 238.992,A -85,B 0,C 180,E1 28428.305,E2 28428.305} C_VEL
LIN {X 0,Y 592.029,Z 238.992,A -85,B 0,C 180,E1 28425.224,E2 28425.224} C_VEL
LIN {X 0,Y 591.957,Z 238.992,A -85,B 0,C 180,E1 28422.197,E2 28422.197} C_VEL
LIN {X 0,Y 592.024,Z 238.99,A -85,B 0,C 180,E1 28419.055,E2 28419.055} C_VEL
LIN {X 0,Y 591.961,Z 238.992,A -85,B 0,C 180,E1 28416.029,E2 28416.029} C_VEL
LIN {X 0,Y 592.013,Z 238.99,A -85,B 0,C 180,E1 28412.87,E2 28412.87} C_VEL
LIN {X 0,Y 591.966,Z 238.992,A -85,B 0,C 180,E1 28409.856,E2 28409.856} C_VEL
LIN {X 0,Y 591.993,Z 238.99,A -85,B 0,C 180,E1 28406.591,E2 28406.591} C_VEL
LIN {X 0,Y 591.974,Z 238.992,A -85,B 0,C 180,E1 28403.672,E2 28403.672} C_VEL
LIN {X 0,Y 591.98,Z 238.99,A -85,B 0,C 180,E1 28400.324,E2 28400.324} C_VEL
LIN {X 0,Y 591.989,Z 238.993,A -85,B 0,C 180,E1 28397.423,E2 28397.423} C_VEL
LIN {X 0,Y 591.976,Z 238.991,A -85,B 0,C 180,E1 28394.124,E2 28394.124} C_VEL
LIN {X 0,Y 592.022,Z 238.994,A -85,B 0,C 180,E1 28391.068,E2 28391.068} C_VEL
LIN {X 0,Y 591.974,Z 238.994,A -85,B 0,C 180,E1 28387.929,E2 28387.929} C_VEL
LIN {X 0,Y 592.005,Z 239.224,A -85,B 0,C 180,E1 28387.656,E2 28387.656} C_VEL
LIN {X 0,Y 594.221,Z 244.847,A -85,B 0,C 180,E1 28387.101,E2 28387.101} C_VEL
LIN {X 0,Y 593.903,Z 289.416,A -85,B 0,C 180,E1 28384.097,E2 28384.097} C_VEL
LIN {X 0,Y 593.912,Z 303.129,A -85,B 0,C 180,E1 28383.217,E2 28383.217} C_VEL
LIN {X 0,Y 594.412,Z 307.424,A -85,B 0,C 180,E1 28383.125,E2 28383.125} C_VEL
LIN {X 0,Y 593.972,Z 528.378,A -85,B 0,C 180,E1 28380.079,E2 28380.079} C_VEL
LIN {X 0,Y 593.813,Z 608.822,A -85,B 0,C 180,E1 28378.962,E2 28378.962} C_VEL
LIN {X 0,Y 593.691,Z 629.751,A -85,B 0,C 180,E1 28378.491,E2 28378.491} C_VEL
LIN {X 0,Y 593.534,Z 650.466,A -85,B 0,C 180,E1 28377.863,E2 28377.863} C_VEL
LIN {X 0,Y 593.399,Z 669.611,A -85,B 0,C 180,E1 28377.114,E2 28377.114} C_VEL
LIN {X 0,Y 593.182,Z 690.774,A -85,B 0,C 180,E1 28376.098,E2 28376.098} C_VEL
LIN {X 0,Y 593.004,Z 710.124,A -85,B 0,C 180,E1 28374.983,E2 28374.983} C_VEL
LIN {X 0,Y 592.808,Z 728.655,A -85,B 0,C 180,E1 28373.713,E2 28373.713} C_VEL
LIN {X 0,Y 592.6,Z 746.892,A -85,B 0,C 180,E1 28372.257,E2 28372.257} C_VEL
LIN {X 0,Y 592.422,Z 764.168,A -85,B 0,C 180,E1 28370.654,E2 28370.654} C_VEL
LIN {X 0,Y 592.292,Z 779.476,A -85,B 0,C 180,E1 28369.013,E2 28369.013} C_VEL
LIN {X 0,Y 592.178,Z 794.121,A -85,B 0,C 180,E1 28367.185,E2 28367.185} C_VEL
LIN {X 0,Y 592.081,Z 806.605,A -85,B 0,C 180,E1 28365.365,E2 28365.365} C_VEL
LIN {X 0,Y 592.006,Z 818.257,A -85,B 0,C 180,E1 28363.377,E2 28363.377} C_VEL
LIN {X 0,Y 591.959,Z 827.529,A -85,B 0,C 180,E1 28361.495,E2 28361.495} C_VEL
LIN {X 0,Y 591.927,Z 835.468,A -85,B 0,C 180,E1 28359.527,E2 28359.527} C_VEL
LIN {X 0,Y 591.919,Z 841.875,A -85,B 0,C 180,E1 28357.57,E2 28357.57} C_VEL
LIN {X 0,Y 591.917,Z 846.811,A -85,B 0,C 180,E1 28355.524,E2 28355.524} C_VEL
LIN {X 0,Y 591.917,Z 850.399,A -85,B 0,C 180,E1 28353.334,E2 28353.334} C_VEL
LIN {X 0,Y 591.908,Z 852.21,A -85,B 0,C 180,E1 28351.257,E2 28351.257} C_VEL
LIN {X 0,Y 591.903,Z 852.328,A -85,B 0,C 180,E1 28349.225,E2 28349.225} C_VEL
LIN {X 0,Y 591.911,Z 850.894,A -85,B 0,C 180,E1 28347.094,E2 28347.094} C_VEL
LIN {X 0,Y 591.916,Z 847.984,A -85,B 0,C 180,E1 28345.057,E2 28345.057} C_VEL
LIN {X 0,Y 591.924,Z 843.396,A -85,B 0,C 180,E1 28343.014,E2 28343.014} C_VEL
LIN {X 0,Y 591.941,Z 837.235,A -85,B 0,C 180,E1 28340.961,E2 28340.961} C_VEL
LIN {X 0,Y 591.951,Z 829.654,A -85,B 0,C 180,E1 28338.996,E2 28338.996} C_VEL
LIN {X 0,Y 591.989,Z 820.324,A -85,B 0,C 180,E1 28337.018,E2 28337.018} C_VEL
LIN {X 0,Y 592.056,Z 809.737,A -85,B 0,C 180,E1 28335.125,E2 28335.125} C_VEL
LIN {X 0,Y 592.126,Z 797.738,A -85,B 0,C 180,E1 28333.317,E2 28333.317} C_VEL
LIN {X 0,Y 592.255,Z 783.71,A -85,B 0,C 180,E1 28331.494,E2 28331.494} C_VEL
LIN {X 0,Y 592.401,Z 768.509,A -85,B 0,C 180,E1 28329.788,E2 28329.788} C_VEL
LIN {X 0,Y 592.566,Z 752.254,A -85,B 0,C 180,E1 28328.209,E2 28328.209} C_VEL
LIN {X 0,Y 592.719,Z 734.776,A -85,B 0,C 180,E1 28326.75,E2 28326.75} C_VEL
LIN {X 0,Y 592.933,Z 715.727,A -85,B 0,C 180,E1 28325.385,E2 28325.385} C_VEL
LIN {X 0,Y 593.152,Z 696.699,A -85,B 0,C 180,E1 28324.22,E2 28324.22} C_VEL
LIN {X 0,Y 593.301,Z 676.786,A -85,B 0,C 180,E1 28323.204,E2 28323.204} C_VEL
LIN {X 0,Y 593.501,Z 655.484,A -85,B 0,C 180,E1 28322.321,E2 28322.321} C_VEL
LIN {X 0,Y 593.684,Z 634.513,A -85,B 0,C 180,E1 28321.634,E2 28321.634} C_VEL
LIN {X 0,Y 593.771,Z 614.053,A -85,B 0,C 180,E1 28321.143,E2 28321.143} C_VEL
LIN {X 0,Y 593.883,Z 586.292,A -85,B 0,C 180,E1 28320.706,E2 28320.706} C_VEL
LIN {X 0,Y 594.266,Z 362.41,A -85,B 0,C 180,E1 28317.64,E2 28317.64} C_VEL
LIN {X 0,Y 594.211,Z 304.603,A -85,B 0,C 180,E1 28316.823,E2 28316.823} C_VEL
LIN {X 0,Y 593.806,Z 302.163,A -85,B 0,C 180,E1 28316.743,E2 28316.743} C_VEL
LIN {X 0,Y 594.072,Z 258.898,A -85,B 0,C 180,E1 28313.855,E2 28313.855} C_VEL
LIN {X 0,Y 594.22,Z 244.849,A -85,B 0,C 180,E1 28312.899,E2 28312.899} C_VEL
LIN {X 0,Y 591.971,Z 238.995,A -85,B 0,C 180,E1 28312.306,E2 28312.306} C_VEL
LIN {X 0,Y 592.041,Z 238.992,A -85,B 0,C 180,E1 28309.165,E2 28309.165} C_VEL
LIN {X 0,Y 591.968,Z 238.992,A -85,B 0,C 180,E1 28306.036,E2 28306.036} C_VEL
LIN {X 0,Y 592.014,Z 238.994,A -85,B 0,C 180,E1 28302.862,E2 28302.862} C_VEL
LIN {X 0,Y 591.965,Z 238.992,A -85,B 0,C 180,E1 28299.93,E2 28299.93} C_VEL
LIN {X 0,Y 592.016,Z 238.993,A -85,B 0,C 180,E1 28296.818,E2 28296.818} C_VEL
LIN {X 0,Y 591.961,Z 238.992,A -85,B 0,C 180,E1 28293.876,E2 28293.876} C_VEL
LIN {X 0,Y 592.009,Z 238.994,A -85,B 0,C 180,E1 28290.721,E2 28290.721} C_VEL
LIN {X 0,Y 591.958,Z 238.993,A -85,B 0,C 180,E1 28287.739,E2 28287.739} C_VEL
LIN {X 0,Y 591.992,Z 238.994,A -85,B 0,C 180,E1 28284.551,E2 28284.551} C_VEL
LIN {X 0,Y 591.952,Z 238.994,A -85,B 0,C 180,E1 28281.711,E2 28281.711} C_VEL
LIN {X 0,Y 591.994,Z 238.996,A -85,B 0,C 180,E1 28278.514,E2 28278.514} C_VEL
LIN {X 0,Y 591.973,Z 239.133,A -85,B 0,C 180,E1 28278.068,E2 28278.068} C_VEL
LIN {X 0,Y 593.263,Z 242.489,A -85,B 0,C 180,E1 28277.939,E2 28277.939} C_VEL
LIN {X 0,Y 594.343,Z 244.264,A -85,B 0,C 180,E1 28277.846,E2 28277.846} C_VEL
LIN {X 0,Y 593.911,Z 481.765,A -85,B 0,C 180,E1 28274.581,E2 28274.581} C_VEL
LIN {X 0,Y 593.798,Z 529.976,A -85,B 0,C 180,E1 28273.897,E2 28273.897} C_VEL
LIN {X 0,Y 593.7,Z 551.217,A -85,B 0,C 180,E1 28273.409,E2 28273.409} C_VEL
LIN {X 0,Y 593.507,Z 573.57,A -85,B 0,C 180,E1 28272.706,E2 28272.706} C_VEL
LIN {X 0,Y 593.344,Z 594.391,A -85,B 0,C 180,E1 28271.865,E2 28271.865} C_VEL
LIN {X 0,Y 593.164,Z 614.868,A -85,B 0,C 180,E1 28270.834,E2 28270.834} C_VEL
LIN {X 0,Y 592.944,Z 634.377,A -85,B 0,C 180,E1 28269.66,E2 28269.66} C_VEL
LIN {X 0,Y 592.752,Z 653.045,A -85,B 0,C 180,E1 28268.342,E2 28268.342} C_VEL
LIN {X 0,Y 592.579,Z 671.293,A -85,B 0,C 180,E1 28266.833,E2 28266.833} C_VEL
LIN {X 0,Y 592.403,Z 687.895,A -85,B 0,C 180,E1 28265.23,E2 28265.23} C_VEL
LIN {X 0,Y 592.258,Z 702.701,A -85,B 0,C 180,E1 28263.582,E2 28263.582} C_VEL
LIN {X 0,Y 592.146,Z 717.004,A -85,B 0,C 180,E1 28261.743,E2 28261.743} C_VEL
LIN {X 0,Y 592.065,Z 729.87,A -85,B 0,C 180,E1 28259.808,E2 28259.808} C_VEL
LIN {X 0,Y 591.995,Z 740.668,A -85,B 0,C 180,E1 28257.872,E2 28257.872} C_VEL
LIN {X 0,Y 591.952,Z 750.166,A -85,B 0,C 180,E1 28255.836,E2 28255.836} C_VEL
LIN {X 0,Y 591.933,Z 757.941,A -85,B 0,C 180,E1 28253.795,E2 28253.795} C_VEL
LIN {X 0,Y 591.919,Z 763.911,A -85,B 0,C 180,E1 28251.746,E2 28251.746} C_VEL
LIN {X 0,Y 591.917,Z 766.826,A -85,B 0,C 180,E1 28250.474,E2 28250.474} C_VEL
LIN {X 0,Y 590.923,Z 768.288,A -85,B 0,C 180,E1 28249.742,E2 28249.742} C_VEL
LIN {X 0,Y 584.571,Z 771.134,A -85,B 0,C 180,E1 28247.722,E2 28247.722} C_VEL
LIN {X 0,Y 583.911,Z 771.614,A -85,B 0,C 180,E1 28247.126,E2 28247.126} C_VEL
LIN {X 0,Y 583.917,Z 772.5,A -85,B 0,C 180,E1 28244.963,E2 28244.963} C_VEL
LIN {X 0,Y 583.915,Z 771.652,A -85,B 0,C 180,E1 28242.841,E2 28242.841} C_VEL
LIN {X 0,Y 583.914,Z 769.051,A -85,B 0,C 180,E1 28240.6,E2 28240.6} C_VEL
LIN {X 0,Y 583.912,Z 765.02,A -85,B 0,C 180,E1 28238.506,E2 28238.506} C_VEL
LIN {X 0,Y 583.921,Z 759.469,A -85,B 0,C 180,E1 28236.488,E2 28236.488} C_VEL
LIN {X 0,Y 583.959,Z 751.839,A -85,B 0,C 180,E1 28234.332,E2 28234.332} C_VEL
LIN {X 0,Y 584.018,Z 743.197,A -85,B 0,C 180,E1 28232.359,E2 28232.359} C_VEL
LIN {X 0,Y 584.096,Z 732.5,A -85,B 0,C 180,E1 28230.352,E2 28230.352} C_VEL
LIN {X 0,Y 584.23,Z 719.59,A -85,B 0,C 180,E1 28228.307,E2 28228.307} C_VEL
LIN {X 0,Y 584.42,Z 705.89,A -85,B 0,C 180,E1 28226.457,E2 28226.457} C_VEL
LIN {X 0,Y 584.635,Z 690.442,A -85,B 0,C 180,E1 28224.665,E2 28224.665} C_VEL
LIN {X 0,Y 584.885,Z 673.418,A -85,B 0,C 180,E1 28222.972,E2 28222.972} C_VEL
LIN {X 0,Y 585.135,Z 656.218,A -85,B 0,C 180,E1 28221.501,E2 28221.501} C_VEL
LIN {X 0,Y 585.457,Z 637.39,A -85,B 0,C 180,E1 28220.115,E2 28220.115} C_VEL
LIN {X 0,Y 585.774,Z 618.339,A -85,B 0,C 180,E1 28218.92,E2 28218.92} C_VEL
LIN {X 0,Y 586.032,Z 598.107,A -85,B 0,C 180,E1 28217.863,E2 28217.863} C_VEL
LIN {X 0,Y 586.337,Z 576.933,A -85,B 0,C 180,E1 28216.961,E2 28216.961} C_VEL
LIN {X 0,Y 586.587,Z 555.58,A -85,B 0,C 180,E1 28216.244,E2 28216.244} C_VEL
LIN {X 0,Y 586.738,Z 534.158,A -85,B 0,C 180,E1 28215.719,E2 28215.719} C_VEL
LIN {X 0,Y 586.898,Z 507.426,A -85,B 0,C 180,E1 28215.293,E2 28215.293} C_VEL
LIN {X 0,Y 587.555,Z 276.444,A -85,B 0,C 180,E1 28212.094,E2 28212.094} C_VEL
LIN {X 0,Y 587.482,Z 246.998,A -85,B 0,C 180,E1 28211.669,E2 28211.669} C_VEL
LIN {X 0,Y 584.318,Z 241.1,A -85,B 0,C 180,E1 28211.38,E2 28211.38} C_VEL
LIN {X 0,Y 584.096,Z 239.981,A -85,B 0,C 180,E1 28211.322,E2 28211.322} C_VEL
LIN {X 0,Y 584.059,Z 239.97,A -85,B 0,C 180,E1 28208.171,E2 28208.171} C_VEL
LIN {X 0,Y 584.087,Z 239.982,A -85,B 0,C 180,E1 28204.873,E2 28204.873} C_VEL
LIN {X 0,Y 584.092,Z 239.974,A -85,B 0,C 180,E1 28201.589,E2 28201.589} C_VEL
LIN {X 0,Y 584.057,Z 239.979,A -85,B 0,C 180,E1 28198.372,E2 28198.372} C_VEL
LIN {X 0,Y 584.098,Z 239.977,A -85,B 0,C 180,E1 28195.23,E2 28195.23} C_VEL
LIN {X 0,Y 584.052,Z 239.977,A -85,B 0,C 180,E1 28192.02,E2 28192.02} C_VEL
LIN {X 0,Y 584.091,Z 239.982,A -85,B 0,C 180,E1 28188.774,E2 28188.774} C_VEL
LIN {X 0,Y 584.066,Z 239.975,A -85,B 0,C 180,E1 28185.592,E2 28185.592} C_VEL
LIN {X 0,Y 584.056,Z 239.979,A -85,B 0,C 180,E1 28182.257,E2 28182.257} C_VEL
LIN {X 0,Y 584.099,Z 239.976,A -85,B 0,C 180,E1 28179.062,E2 28179.062} C_VEL
LIN {X 0,Y 584.046,Z 239.977,A -85,B 0,C 180,E1 28175.897,E2 28175.897} C_VEL
LIN {X 0,Y 584.098,Z 239.979,A -85,B 0,C 180,E1 28172.748,E2 28172.748} C_VEL
LIN {X 0,Y 584.047,Z 239.976,A -85,B 0,C 180,E1 28169.609,E2 28169.609} C_VEL
LIN {X 0,Y 584.076,Z 239.979,A -85,B 0,C 180,E1 28166.347,E2 28166.347} C_VEL
LIN {X 0,Y 584.063,Z 239.976,A -85,B 0,C 180,E1 28163.217,E2 28163.217} C_VEL
LIN {X 0,Y 584.049,Z 239.979,A -85,B 0,C 180,E1 28159.945,E2 28159.945} C_VEL
LIN {X 0,Y 584.091,Z 239.975,A -85,B 0,C 180,E1 28156.841,E2 28156.841} C_VEL
LIN {X 0,Y 584.04,Z 239.979,A -85,B 0,C 180,E1 28153.695,E2 28153.695} C_VEL
LIN {X 0,Y 584.101,Z 239.977,A -85,B 0,C 180,E1 28150.587,E2 28150.587} C_VEL
LIN {X 0,Y 584.036,Z 239.979,A -85,B 0,C 180,E1 28147.452,E2 28147.452} C_VEL
LIN {X 0,Y 584.098,Z 239.981,A -85,B 0,C 180,E1 28144.338,E2 28144.338} C_VEL
LIN {X 0,Y 584.036,Z 239.978,A -85,B 0,C 180,E1 28141.222,E2 28141.222} C_VEL
LIN {X 0,Y 584.079,Z 239.981,A -85,B 0,C 180,E1 28138.066,E2 28138.066} C_VEL
LIN {X 0,Y 584.038,Z 239.979,A -85,B 0,C 180,E1 28135.006,E2 28135.006} C_VEL
LIN {X 0,Y 584.044,Z 239.981,A -85,B 0,C 180,E1 28131.631,E2 28131.631} C_VEL
LIN {X 0,Y 584.057,Z 239.978,A -85,B 0,C 180,E1 28128.641,E2 28128.641} C_VEL
LIN {X 0,Y 584.034,Z 239.981,A -85,B 0,C 180,E1 28125.41,E2 28125.41} C_VEL
LIN {X 0,Y 584.071,Z 239.979,A -85,B 0,C 180,E1 28122.411,E2 28122.411} C_VEL
LIN {X 0,Y 584.029,Z 239.98,A -85,B 0,C 180,E1 28119.302,E2 28119.302} C_VEL
LIN {X 0,Y 584.069,Z 239.98,A -85,B 0,C 180,E1 28116.319,E2 28116.319} C_VEL
LIN {X 0,Y 584.024,Z 239.981,A -85,B 0,C 180,E1 28113.16,E2 28113.16} C_VEL
LIN {X 0,Y 584.085,Z 239.979,A -85,B 0,C 180,E1 28110.101,E2 28110.101} C_VEL
LIN {X 0,Y 584.02,Z 239.981,A -85,B 0,C 180,E1 28106.978,E2 28106.978} C_VEL
LIN {X 0,Y 584.09,Z 239.98,A -85,B 0,C 180,E1 28103.924,E2 28103.924} C_VEL
LIN {X 0,Y 584.017,Z 239.981,A -85,B 0,C 180,E1 28100.813,E2 28100.813} C_VEL
LIN {X 0,Y 584.091,Z 239.982,A -85,B 0,C 180,E1 28097.739,E2 28097.739} C_VEL
LIN {X 0,Y 584.014,Z 239.981,A -85,B 0,C 180,E1 28094.676,E2 28094.676} C_VEL
LIN {X 0,Y 584.081,Z 239.981,A -85,B 0,C 180,E1 28091.552,E2 28091.552} C_VEL
LIN {X 0,Y 584.013,Z 239.982,A -85,B 0,C 180,E1 28088.465,E2 28088.465} C_VEL
LIN {X 0,Y 584.057,Z 239.982,A -85,B 0,C 180,E1 28085.303,E2 28085.303} C_VEL
LIN {X 0,Y 584.013,Z 239.982,A -85,B 0,C 180,E1 28082.354,E2 28082.354} C_VEL
LIN {X 0,Y 584.058,Z 239.982,A -85,B 0,C 180,E1 28079.214,E2 28079.214} C_VEL
LIN {X 0,Y 584.015,Z 239.982,A -85,B 0,C 180,E1 28076.269,E2 28076.269} C_VEL
LIN {X 0,Y 584.06,Z 239.981,A -85,B 0,C 180,E1 28073.116,E2 28073.116} C_VEL
LIN {X 0,Y 584.021,Z 239.982,A -85,B 0,C 180,E1 28070.141,E2 28070.141} C_VEL
LIN {X 0,Y 584.05,Z 239.98,A -85,B 0,C 180,E1 28066.922,E2 28066.922} C_VEL
LIN {X 0,Y 584.021,Z 239.981,A -85,B 0,C 180,E1 28064.101,E2 28064.101} C_VEL
LIN {X 0,Y 584.06,Z 239.98,A -85,B 0,C 180,E1 28060.899,E2 28060.899} C_VEL
LIN {X 0,Y 584.025,Z 239.981,A -85,B 0,C 180,E1 28057.979,E2 28057.979} C_VEL
LIN {X 0,Y 584.056,Z 239.979,A -85,B 0,C 180,E1 28054.768,E2 28054.768} C_VEL
LIN {X 0,Y 584.031,Z 239.981,A -85,B 0,C 180,E1 28051.802,E2 28051.802} C_VEL
LIN {X 0,Y 584.041,Z 239.98,A -85,B 0,C 180,E1 28048.488,E2 28048.488} C_VEL
LIN {X 0,Y 584.042,Z 239.982,A -85,B 0,C 180,E1 28045.601,E2 28045.601} C_VEL
LIN {X 0,Y 584.036,Z 239.979,A -85,B 0,C 180,E1 28042.27,E2 28042.27} C_VEL
LIN {X 0,Y 584.066,Z 239.982,A -85,B 0,C 180,E1 28039.289,E2 28039.289} C_VEL
LIN {X 0,Y 584.034,Z 239.981,A -85,B 0,C 180,E1 28036.103,E2 28036.103} C_VEL
LIN {X 0,Y 584.087,Z 239.983,A -85,B 0,C 180,E1 28033.033,E2 28033.033} C_VEL
LIN {X 0,Y 584.033,Z 239.98,A -85,B 0,C 180,E1 28029.917,E2 28029.917} C_VEL
LIN {X 0,Y 584.068,Z 240.114,A -85,B 0,C 180,E1 28028.196,E2 28028.196} C_VEL
LIN {X 0,Y 586.765,Z 246.855,A -85,B 0,C 180,E1 28027.512,E2 28027.512} C_VEL
LIN {X 0,Y 587.38,Z 249.237,A -85,B 0,C 180,E1 28027.299,E2 28027.299} C_VEL
LIN {X 0,Y 586.901,Z 292.91,A -85,B 0,C 180,E1 28024.324,E2 28024.324} C_VEL
LIN {X 0,Y 586.912,Z 303.196,A -85,B 0,C 180,E1 28023.665,E2 28023.665} C_VEL
LIN {X 0,Y 587.705,Z 308.517,A -85,B 0,C 180,E1 28023.537,E2 28023.537} C_VEL
LIN {X 0,Y 587.045,Z 529.117,A -85,B 0,C 180,E1 28020.461,E2 28020.461} C_VEL
LIN {X 0,Y 586.805,Z 608.929,A -85,B 0,C 180,E1 28019.339,E2 28019.339} C_VEL
LIN {X 0,Y 586.616,Z 630.049,A -85,B 0,C 180,E1 28018.859,E2 28018.859} C_VEL
LIN {X 0,Y 586.368,Z 651.796,A -85,B 0,C 180,E1 28018.184,E2 28018.184} C_VEL
LIN {X 0,Y 586.153,Z 672.16,A -85,B 0,C 180,E1 28017.367,E2 28017.367} C_VEL
LIN {X 0,Y 585.832,Z 692.468,A -85,B 0,C 180,E1 28016.358,E2 28016.358} C_VEL
LIN {X 0,Y 585.52,Z 712.551,A -85,B 0,C 180,E1 28015.162,E2 28015.162} C_VEL
LIN {X 0,Y 585.25,Z 731.471,A -85,B 0,C 180,E1 28013.83,E2 28013.83} C_VEL
LIN {X 0,Y 584.944,Z 749.105,A -85,B 0,C 180,E1 28012.37,E2 28012.37} C_VEL
LIN {X 0,Y 584.679,Z 765.687,A -85,B 0,C 180,E1 28010.783,E2 28010.783} C_VEL
LIN {X 0,Y 584.466,Z 781.177,A -85,B 0,C 180,E1 28009.07,E2 28009.07} C_VEL
LIN {X 0,Y 584.311,Z 795.151,A -85,B 0,C 180,E1 28007.286,E2 28007.286} C_VEL
LIN {X 0,Y 584.163,Z 807.836,A -85,B 0,C 180,E1 28005.384,E2 28005.384} C_VEL
LIN {X 0,Y 584.051,Z 819.296,A -85,B 0,C 180,E1 28003.361,E2 28003.361} C_VEL
LIN {X 0,Y 583.988,Z 828.847,A -85,B 0,C 180,E1 28001.354,E2 28001.354} C_VEL
LIN {X 0,Y 583.945,Z 836.533,A -85,B 0,C 180,E1 27999.36,E2 27999.36} C_VEL
LIN {X 0,Y 583.927,Z 843.147,A -85,B 0,C 180,E1 27997.18,E2 27997.18} C_VEL
LIN {X 0,Y 583.919,Z 847.826,A -85,B 0,C 180,E1 27995.107,E2 27995.107} C_VEL
LIN {X 0,Y 583.916,Z 850.785,A -85,B 0,C 180,E1 27993.042,E2 27993.042} C_VEL
LIN {X 0,Y 583.909,Z 852.307,A -85,B 0,C 180,E1 27990.882,E2 27990.882} C_VEL
LIN {X 0,Y 583.912,Z 852.239,A -85,B 0,C 180,E1 27988.822,E2 27988.822} C_VEL
LIN {X 0,Y 583.917,Z 850.558,A -85,B 0,C 180,E1 27986.76,E2 27986.76} C_VEL
LIN {X 0,Y 583.918,Z 847.218,A -85,B 0,C 180,E1 27984.595,E2 27984.595} C_VEL
LIN {X 0,Y 583.921,Z 842.633,A -85,B 0,C 180,E1 27982.621,E2 27982.621} C_VEL
LIN {X 0,Y 583.941,Z 836.003,A -85,B 0,C 180,E1 27980.491,E2 27980.491} C_VEL
LIN {X 0,Y 583.988,Z 828.427,A -85,B 0,C 180,E1 27978.544,E2 27978.544} C_VEL
LIN {X 0,Y 584.05,Z 818.767,A -85,B 0,C 180,E1 27976.536,E2 27976.536} C_VEL
LIN {X 0,Y 584.164,Z 807.107,A -85,B 0,C 180,E1 27974.501,E2 27974.501} C_VEL
LIN {X 0,Y 584.312,Z 794.874,A -85,B 0,C 180,E1 27972.677,E2 27972.677} C_VEL
LIN {X 0,Y 584.482,Z 780.31,A -85,B 0,C 180,E1 27970.825,E2 27970.825} C_VEL
LIN {X 0,Y 584.686,Z 765.161,A -85,B 0,C 180,E1 27969.163,E2 27969.163} C_VEL
LIN {X 0,Y 584.961,Z 747.473,A -85,B 0,C 180,E1 27967.487,E2 27967.487} C_VEL
LIN {X 0,Y 585.267,Z 730.011,A -85,B 0,C 180,E1 27966.062,E2 27966.062} C_VEL
LIN {X 0,Y 585.543,Z 711.713,A -85,B 0,C 180,E1 27964.783,E2 27964.783} C_VEL
LIN {X 0,Y 585.838,Z 691.734,A -85,B 0,C 180,E1 27963.602,E2 27963.602} C_VEL
LIN {X 0,Y 586.154,Z 672.11,A -85,B 0,C 180,E1 27962.631,E2 27962.631} C_VEL
LIN {X 0,Y 586.372,Z 651.74,A -85,B 0,C 180,E1 27961.814,E2 27961.814} C_VEL
LIN {X 0,Y 586.62,Z 629.843,A -85,B 0,C 180,E1 27961.136,E2 27961.136} C_VEL
LIN {X 0,Y 586.81,Z 608.689,A -85,B 0,C 180,E1 27960.657,E2 27960.657} C_VEL
LIN {X 0,Y 587.077,Z 519.826,A -85,B 0,C 180,E1 27959.412,E2 27959.412} C_VEL
LIN {X 0,Y 587.696,Z 307.083,A -85,B 0,C 180,E1 27956.442,E2 27956.442} C_VEL
LIN {X 0,Y 586.795,Z 302.112,A -85,B 0,C 180,E1 27956.289,E2 27956.289} C_VEL
LIN {X 0,Y 587.225,Z 259.684,A -85,B 0,C 180,E1 27953.42,E2 27953.42} C_VEL
LIN {X 0,Y 587.2,Z 247.769,A -85,B 0,C 180,E1 27952.585,E2 27952.585} C_VEL
LIN {X 0,Y 584.084,Z 240.229,A -85,B 0,C 180,E1 27951.814,E2 27951.814} C_VEL
LIN {X 0,Y 584.072,Z 239.984,A -85,B 0,C 180,E1 27948.871,E2 27948.871} C_VEL
LIN {X 0,Y 584.038,Z 239.981,A -85,B 0,C 180,E1 27945.831,E2 27945.831} C_VEL
LIN {X 0,Y 584.036,Z 239.982,A -85,B 0,C 180,E1 27942.45,E2 27942.45} C_VEL
LIN {X 0,Y 584.048,Z 239.981,A -85,B 0,C 180,E1 27939.557,E2 27939.557} C_VEL
LIN {X 0,Y 584.029,Z 239.982,A -85,B 0,C 180,E1 27936.325,E2 27936.325} C_VEL
LIN {X 0,Y 584.047,Z 239.981,A -85,B 0,C 180,E1 27933.453,E2 27933.453} C_VEL
LIN {X 0,Y 584.021,Z 239.982,A -85,B 0,C 180,E1 27930.166,E2 27930.166} C_VEL
LIN {X 0,Y 584.078,Z 239.982,A -85,B 0,C 180,E1 27927.088,E2 27927.088} C_VEL
LIN {X 0,Y 584.013,Z 239.983,A -85,B 0,C 180,E1 27923.939,E2 27923.939} C_VEL
LIN {X 0,Y 584.088,Z 239.982,A -85,B 0,C 180,E1 27920.826,E2 27920.826} C_VEL
LIN {X 0,Y 584.093,Z 240.217,A -85,B 0,C 180,E1 27918.558,E2 27918.558} C_VEL
LIN {X 0,Y 585.473,Z 243.647,A -85,B 0,C 180,E1 27918.418,E2 27918.418} C_VEL
LIN {X 0,Y 587.617,Z 247.444,A -85,B 0,C 180,E1 27918.226,E2 27918.226} C_VEL
LIN {X 0,Y 586.949,Z 484.314,A -85,B 0,C 180,E1 27914.933,E2 27914.933} C_VEL
LIN {X 0,Y 586.785,Z 530.083,A -85,B 0,C 180,E1 27914.274,E2 27914.274} C_VEL
LIN {X 0,Y 586.626,Z 551.582,A -85,B 0,C 180,E1 27913.775,E2 27913.775} C_VEL
LIN {X 0,Y 586.347,Z 573.327,A -85,B 0,C 180,E1 27913.084,E2 27913.084} C_VEL
LIN {X 0,Y 586.102,Z 594.628,A -85,B 0,C 180,E1 27912.213,E2 27912.213} C_VEL
LIN {X 0,Y 585.815,Z 615.102,A -85,B 0,C 180,E1 27911.171,E2 27911.171} C_VEL
LIN {X 0,Y 585.478,Z 634.839,A -85,B 0,C 180,E1 27909.966,E2 27909.966} C_VEL
LIN {X 0,Y 585.189,Z 653.836,A -85,B 0,C 180,E1 27908.599,E2 27908.599} C_VEL
LIN {X 0,Y 584.916,Z 671.985,A -85,B 0,C 180,E1 27907.071,E2 27907.071} C_VEL
LIN {X 0,Y 584.655,Z 688.99,A -85,B 0,C 180,E1 27905.398,E2 27905.398} C_VEL
LIN {X 0,Y 584.427,Z 704.437,A -85,B 0,C 180,E1 27903.631,E2 27903.631} C_VEL
LIN {X 0,Y 584.255,Z 718.457,A -85,B 0,C 180,E1 27901.766,E2 27901.766} C_VEL
LIN {X 0,Y 584.138,Z 730.526,A -85,B 0,C 180,E1 27899.903,E2 27899.903} C_VEL
LIN {X 0,Y 584.038,Z 741.237,A -85,B 0,C 180,E1 27897.941,E2 27897.941} C_VEL
LIN {X 0,Y 583.973,Z 750.613,A -85,B 0,C 180,E1 27895.878,E2 27895.878} C_VEL
LIN {X 0,Y 583.942,Z 758.283,A -85,B 0,C 180,E1 27893.809,E2 27893.809} C_VEL
LIN {X 0,Y 583.923,Z 764.193,A -85,B 0,C 180,E1 27891.732,E2 27891.732} C_VEL
LIN {X 0,Y 583.91,Z 768.673,A -85,B 0,C 180,E1 27889.544,E2 27889.544} C_VEL
LIN {X 0,Y 583.906,Z 771.395,A -85,B 0,C 180,E1 27887.435,E2 27887.435} C_VEL
LIN {X 0,Y 583.911,Z 771.614,A -85,B 0,C 180,E1 27887.126,E2 27887.126} C_VEL
LIN {X 0,Y 582.896,Z 772.134,A -85,B 0,C 180,E1 27886.371,E2 27886.371} C_VEL
LIN {X 0,Y 576.557,Z 772.42,A -85,B 0,C 180,E1 27884.304,E2 27884.304} C_VEL
LIN {X 0,Y 575.913,Z 772.22,A -85,B 0,C 180,E1 27883.698,E2 27883.698} C_VEL
LIN {X 0,Y 575.914,Z 770.467,A -85,B 0,C 180,E1 27881.582,E2 27881.582} C_VEL
LIN {X 0,Y 575.921,Z 766.973,A -85,B 0,C 180,E1 27879.352,E2 27879.352} C_VEL
LIN {X 0,Y 575.933,Z 761.938,A -85,B 0,C 180,E1 27877.199,E2 27877.199} C_VEL
LIN {X 0,Y 575.963,Z 755.481,A -85,B 0,C 180,E1 27875.161,E2 27875.161} C_VEL
LIN {X 0,Y 576.031,Z 747.207,A -85,B 0,C 180,E1 27873.064,E2 27873.064} C_VEL
LIN {X 0,Y 576.133,Z 737.273,A -85,B 0,C 180,E1 27871.007,E2 27871.007} C_VEL
LIN {X 0,Y 576.255,Z 726.259,A -85,B 0,C 180,E1 27869.099,E2 27869.099} C_VEL
LIN {X 0,Y 576.469,Z 712.917,A -85,B 0,C 180,E1 27867.122,E2 27867.122} C_VEL
LIN {X 0,Y 576.737,Z 698.973,A -85,B 0,C 180,E1 27865.347,E2 27865.347} C_VEL
LIN {X 0,Y 577.06,Z 682.412,A -85,B 0,C 180,E1 27863.539,E2 27863.539} C_VEL
LIN {X 0,Y 577.405,Z 665.402,A -85,B 0,C 180,E1 27861.944,E2 27861.944} C_VEL
LIN {X 0,Y 577.79,Z 646.838,A -85,B 0,C 180,E1 27860.448,E2 27860.448} C_VEL
LIN {X 0,Y 578.233,Z 627.551,A -85,B 0,C 180,E1 27859.122,E2 27859.122} C_VEL
LIN {X 0,Y 578.657,Z 607.173,A -85,B 0,C 180,E1 27857.948,E2 27857.948} C_VEL
LIN {X 0,Y 579.014,Z 586.212,A -85,B 0,C 180,E1 27856.958,E2 27856.958} C_VEL
LIN {X 0,Y 579.395,Z 564.023,A -85,B 0,C 180,E1 27856.126,E2 27856.126} C_VEL
LIN {X 0,Y 579.689,Z 542.01,A -85,B 0,C 180,E1 27855.502,E2 27855.502} C_VEL
LIN {X 0,Y 579.871,Z 520.28,A -85,B 0,C 180,E1 27855.083,E2 27855.083} C_VEL
LIN {X 0,Y 580.764,Z 293.4,A -85,B 0,C 180,E1 27851.906,E2 27851.906} C_VEL
LIN {X 0,Y 580.751,Z 249.681,A -85,B 0,C 180,E1 27851.271,E2 27851.271} C_VEL
LIN {X 0,Y 576.437,Z 242.342,A -85,B 0,C 180,E1 27850.877,E2 27850.877} C_VEL
LIN {X 0,Y 576.139,Z 240.972,A -85,B 0,C 180,E1 27850.833,E2 27850.833} C_VEL
LIN {X 0,Y 576.155,Z 240.95,A -85,B 0,C 180,E1 27847.652,E2 27847.652} C_VEL
LIN {X 0,Y 576.119,Z 240.969,A -85,B 0,C 180,E1 27844.457,E2 27844.457} C_VEL
LIN {X 0,Y 576.159,Z 240.968,A -85,B 0,C 180,E1 27841.185,E2 27841.185} C_VEL
LIN {X 0,Y 576.122,Z 240.966,A -85,B 0,C 180,E1 27837.943,E2 27837.943} C_VEL
LIN {X 0,Y 576.132,Z 240.97,A -85,B 0,C 180,E1 27834.586,E2 27834.586} C_VEL
LIN {X 0,Y 576.158,Z 240.963,A -85,B 0,C 180,E1 27831.373,E2 27831.373} C_VEL
LIN {X 0,Y 576.112,Z 240.967,A -85,B 0,C 180,E1 27828.1,E2 27828.1} C_VEL
LIN {X 0,Y 576.16,Z 240.969,A -85,B 0,C 180,E1 27824.859,E2 27824.859} C_VEL
LIN {X 0,Y 576.115,Z 240.965,A -85,B 0,C 180,E1 27821.717,E2 27821.717} C_VEL
LIN {X 0,Y 576.128,Z 240.969,A -85,B 0,C 180,E1 27818.383,E2 27818.383} C_VEL
LIN {X 0,Y 576.148,Z 240.963,A -85,B 0,C 180,E1 27815.178,E2 27815.178} C_VEL
LIN {X 0,Y 576.109,Z 240.967,A -85,B 0,C 180,E1 27811.99,E2 27811.99} C_VEL
LIN {X 0,Y 576.162,Z 240.965,A -85,B 0,C 180,E1 27808.808,E2 27808.808} C_VEL
LIN {X 0,Y 576.104,Z 240.965,A -85,B 0,C 180,E1 27805.621,E2 27805.621} C_VEL
LIN {X 0,Y 576.152,Z 240.969,A -85,B 0,C 180,E1 27802.422,E2 27802.422} C_VEL
LIN {X 0,Y 576.113,Z 240.966,A -85,B 0,C 180,E1 27799.299,E2 27799.299} C_VEL
LIN {X 0,Y 576.112,Z 240.968,A -85,B 0,C 180,E1 27795.939,E2 27795.939} C_VEL
LIN {X 0,Y 576.143,Z 240.965,A -85,B 0,C 180,E1 27792.842,E2 27792.842} C_VEL
LIN {X 0,Y 576.098,Z 240.968,A -85,B 0,C 180,E1 27789.584,E2 27789.584} C_VEL
LIN {X 0,Y 576.162,Z 240.969,A -85,B 0,C 180,E1 27786.369,E2 27786.369} C_VEL
LIN {X 0,Y 576.1,Z 240.968,A -85,B 0,C 180,E1 27783.178,E2 27783.178} C_VEL
LIN {X 0,Y 576.12,Z 240.97,A -85,B 0,C 180,E1 27779.898,E2 27779.898} C_VEL
LIN {X 0,Y 576.112,Z 240.966,A -85,B 0,C 180,E1 27776.861,E2 27776.861} C_VEL
LIN {X 0,Y 576.101,Z 240.968,A -85,B 0,C 180,E1 27773.592,E2 27773.592} C_VEL
LIN {X 0,Y 576.131,Z 240.968,A -85,B 0,C 180,E1 27770.556,E2 27770.556} C_VEL
LIN {X 0,Y 576.092,Z 240.97,A -85,B 0,C 180,E1 27767.379,E2 27767.379} C_VEL
LIN {X 0,Y 576.157,Z 240.968,A -85,B 0,C 180,E1 27764.234,E2 27764.234} C_VEL
LIN {X 0,Y 576.087,Z 240.97,A -85,B 0,C 180,E1 27761.129,E2 27761.129} C_VEL
LIN {X 0,Y 576.161,Z 240.969,A -85,B 0,C 180,E1 27758.016,E2 27758.016} C_VEL
LIN {X 0,Y 576.084,Z 240.968,A -85,B 0,C 180,E1 27754.94,E2 27754.94} C_VEL
LIN {X 0,Y 576.138,Z 240.97,A -85,B 0,C 180,E1 27751.751,E2 27751.751} C_VEL
LIN {X 0,Y 576.084,Z 240.969,A -85,B 0,C 180,E1 27748.733,E2 27748.733} C_VEL
LIN {X 0,Y 576.115,Z 240.97,A -85,B 0,C 180,E1 27745.491,E2 27745.491} C_VEL
LIN {X 0,Y 576.085,Z 240.97,A -85,B 0,C 180,E1 27742.553,E2 27742.553} C_VEL
LIN {X 0,Y 576.096,Z 240.97,A -85,B 0,C 180,E1 27739.244,E2 27739.244} C_VEL
LIN {X 0,Y 576.093,Z 240.97,A -85,B 0,C 180,E1 27736.312,E2 27736.312} C_VEL
LIN {X 0,Y 576.086,Z 240.971,A -85,B 0,C 180,E1 27733.038,E2 27733.038} C_VEL
LIN {X 0,Y 576.102,Z 240.969,A -85,B 0,C 180,E1 27730.094,E2 27730.094} C_VEL
LIN {X 0,Y 576.078,Z 240.971,A -85,B 0,C 180,E1 27726.877,E2 27726.877} C_VEL
LIN {X 0,Y 576.113,Z 240.971,A -85,B 0,C 180,E1 27723.88,E2 27723.88} C_VEL
LIN {X 0,Y 576.075,Z 240.97,A -85,B 0,C 180,E1 27720.695,E2 27720.695} C_VEL
LIN {X 0,Y 576.126,Z 240.971,A -85,B 0,C 180,E1 27717.711,E2 27717.711} C_VEL
LIN {X 0,Y 576.075,Z 240.97,A -85,B 0,C 180,E1 27714.521,E2 27714.521} C_VEL
LIN {X 0,Y 576.153,Z 240.97,A -85,B 0,C 180,E1 27711.416,E2 27711.416} C_VEL
LIN {X 0,Y 576.077,Z 240.97,A -85,B 0,C 180,E1 27708.282,E2 27708.282} C_VEL
LIN {X 0,Y 576.139,Z 240.969,A -85,B 0,C 180,E1 27705.116,E2 27705.116} C_VEL
LIN {X 0,Y 576.082,Z 240.97,A -85,B 0,C 180,E1 27702.108,E2 27702.108} C_VEL
LIN {X 0,Y 576.131,Z 240.968,A -85,B 0,C 180,E1 27698.945,E2 27698.945} C_VEL
LIN {X 0,Y 576.089,Z 240.969,A -85,B 0,C 180,E1 27695.908,E2 27695.908} C_VEL
LIN {X 0,Y 576.107,Z 240.968,A -85,B 0,C 180,E1 27692.617,E2 27692.617} C_VEL
LIN {X 0,Y 576.1,Z 240.97,A -85,B 0,C 180,E1 27689.665,E2 27689.665} C_VEL
LIN {X 0,Y 576.098,Z 240.969,A -85,B 0,C 180,E1 27686.382,E2 27686.382} C_VEL
LIN {X 0,Y 576.113,Z 240.971,A -85,B 0,C 180,E1 27683.466,E2 27683.466} C_VEL
LIN {X 0,Y 576.094,Z 240.969,A -85,B 0,C 180,E1 27680.176,E2 27680.176} C_VEL
LIN {X 0,Y 576.143,Z 240.972,A -85,B 0,C 180,E1 27677.133,E2 27677.133} C_VEL
LIN {X 0,Y 576.093,Z 240.971,A -85,B 0,C 180,E1 27673.923,E2 27673.923} C_VEL
LIN {X 0,Y 576.162,Z 240.963,A -85,B 0,C 180,E1 27670.728,E2 27670.728} C_VEL
LIN {X 0,Y 576.169,Z 241.046,A -85,B 0,C 180,E1 27668.748,E2 27668.748} C_VEL
LIN {X 0,Y 577.154,Z 243.996,A -85,B 0,C 180,E1 27668.455,E2 27668.455} C_VEL
LIN {X 0,Y 580.575,Z 252.101,A -85,B 0,C 180,E1 27667.608,E2 27667.608} C_VEL
LIN {X 0,Y 579.943,Z 294.657,A -85,B 0,C 180,E1 27664.675,E2 27664.675} C_VEL
LIN {X 0,Y 579.922,Z 303.131,A -85,B 0,C 180,E1 27664.127,E2 27664.127} C_VEL
LIN {X 0,Y 581.028,Z 309.887,A -85,B 0,C 180,E1 27663.954,E2 27663.954} C_VEL
LIN {X 0,Y 580.142,Z 530.42,A -85,B 0,C 180,E1 27660.844,E2 27660.844} C_VEL
LIN {X 0,Y 579.824,Z 609.036,A -85,B 0,C 180,E1 27659.726,E2 27659.726} C_VEL
LIN {X 0,Y 579.568,Z 630.179,A -85,B 0,C 180,E1 27659.24,E2 27659.24} C_VEL
LIN {X 0,Y 579.254,Z 651.792,A -85,B 0,C 180,E1 27658.562,E2 27658.562} C_VEL
LIN {X 0,Y 578.947,Z 672.164,A -85,B 0,C 180,E1 27657.737,E2 27657.737} C_VEL
LIN {X 0,Y 578.525,Z 691.774,A -85,B 0,C 180,E1 27656.756,E2 27656.756} C_VEL
LIN {X 0,Y 578.137,Z 711.74,A -85,B 0,C 180,E1 27655.561,E2 27655.561} C_VEL
LIN {X 0,Y 577.74,Z 730.811,A -85,B 0,C 180,E1 27654.21,E2 27654.21} C_VEL
LIN {X 0,Y 577.326,Z 748.706,A -85,B 0,C 180,E1 27652.717,E2 27652.717} C_VEL
LIN {X 0,Y 576.966,Z 765.841,A -85,B 0,C 180,E1 27651.057,E2 27651.057} C_VEL
LIN {X 0,Y 576.677,Z 781.178,A -85,B 0,C 180,E1 27649.338,E2 27649.338} C_VEL
LIN {X 0,Y 576.446,Z 795.633,A -85,B 0,C 180,E1 27647.461,E2 27647.461} C_VEL
LIN {X 0,Y 576.246,Z 808.477,A -85,B 0,C 180,E1 27645.497,E2 27645.497} C_VEL
LIN {X 0,Y 576.098,Z 819.297,A -85,B 0,C 180,E1 27643.549,E2 27643.549} C_VEL
LIN {X 0,Y 576.012,Z 828.848,A -85,B 0,C 180,E1 27641.514,E2 27641.514} C_VEL
LIN {X 0,Y 575.954,Z 836.534,A -85,B 0,C 180,E1 27639.491,E2 27639.491} C_VEL
LIN {X 0,Y 575.927,Z 843.147,A -85,B 0,C 180,E1 27637.28,E2 27637.28} C_VEL
LIN {X 0,Y 575.92,Z 847.826,A -85,B 0,C 180,E1 27635.179,E2 27635.179} C_VEL
LIN {X 0,Y 575.916,Z 850.785,A -85,B 0,C 180,E1 27633.084,E2 27633.084} C_VEL
LIN {X 0,Y 575.91,Z 852.307,A -85,B 0,C 180,E1 27630.894,E2 27630.894} C_VEL
LIN {X 0,Y 575.911,Z 852.239,A -85,B 0,C 180,E1 27628.805,E2 27628.805} C_VEL
LIN {X 0,Y 575.917,Z 850.558,A -85,B 0,C 180,E1 27626.715,E2 27626.715} C_VEL
LIN {X 0,Y 575.919,Z 847.218,A -85,B 0,C 180,E1 27624.52,E2 27624.52} C_VEL
LIN {X 0,Y 575.927,Z 842.432,A -85,B 0,C 180,E1 27622.438,E2 27622.438} C_VEL
LIN {X 0,Y 575.954,Z 835.817,A -85,B 0,C 180,E1 27620.305,E2 27620.305} C_VEL
LIN {X 0,Y 576.017,Z 827.776,A -85,B 0,C 180,E1 27618.237,E2 27618.237} C_VEL
LIN {X 0,Y 576.107,Z 818.248,A -85,B 0,C 180,E1 27616.244,E2 27616.244} C_VEL
LIN {X 0,Y 576.25,Z 807.184,A -85,B 0,C 180,E1 27614.295,E2 27614.295} C_VEL
LIN {X 0,Y 576.458,Z 794.873,A -85,B 0,C 180,E1 27612.433,E2 27612.433} C_VEL
LIN {X 0,Y 576.699,Z 780.311,A -85,B 0,C 180,E1 27610.555,E2 27610.555} C_VEL
LIN {X 0,Y 576.983,Z 765.16,A -85,B 0,C 180,E1 27608.872,E2 27608.872} C_VEL
LIN {X 0,Y 577.349,Z 747.474,A -85,B 0,C 180,E1 27607.174,E2 27607.174} C_VEL
LIN {X 0,Y 577.746,Z 729.993,A -85,B 0,C 180,E1 27605.729,E2 27605.729} C_VEL
LIN {X 0,Y 578.138,Z 711.709,A -85,B 0,C 180,E1 27604.437,E2 27604.437} C_VEL
LIN {X 0,Y 578.526,Z 691.736,A -85,B 0,C 180,E1 27603.242,E2 27603.242} C_VEL
LIN {X 0,Y 578.946,Z 672.113,A -85,B 0,C 180,E1 27602.261,E2 27602.261} C_VEL
LIN {X 0,Y 579.257,Z 651.738,A -85,B 0,C 180,E1 27601.436,E2 27601.436} C_VEL
LIN {X 0,Y 579.573,Z 629.715,A -85,B 0,C 180,E1 27600.747,E2 27600.747} C_VEL
LIN {X 0,Y 579.83,Z 608.475,A -85,B 0,C 180,E1 27600.265,E2 27600.265} C_VEL
LIN {X 0,Y 580.266,Z 499.512,A -85,B 0,C 180,E1 27598.725,E2 27598.725} C_VEL
LIN {X 0,Y 580.923,Z 308.145,A -85,B 0,C 180,E1 27596.013,E2 27596.013} C_VEL
LIN {X 0,Y 579.82,Z 302.098,A -85,B 0,C 180,E1 27595.827,E2 27595.827} C_VEL
LIN {X 0,Y 580.411,Z 260.558,A -85,B 0,C 180,E1 27592.981,E2 27592.981} C_VEL
LIN {X 0,Y 580.403,Z 251.461,A -85,B 0,C 180,E1 27592.334,E2 27592.334} C_VEL
LIN {X 0,Y 576.197,Z 241.236,A -85,B 0,C 180,E1 27591.268,E2 27591.268} C_VEL
LIN {X 0,Y 576.14,Z 240.972,A -85,B 0,C 180,E1 27590.952,E2 27590.952} C_VEL
LIN {X 0,Y 576.098,Z 240.971,A -85,B 0,C 180,E1 27587.938,E2 27587.938} C_VEL
LIN {X 0,Y 576.111,Z 240.972,A -85,B 0,C 180,E1 27584.637,E2 27584.637} C_VEL
LIN {X 0,Y 576.105,Z 240.97,A -85,B 0,C 180,E1 27581.661,E2 27581.661} C_VEL
LIN {X 0,Y 576.091,Z 240.971,A -85,B 0,C 180,E1 27578.326,E2 27578.326} C_VEL
LIN {X 0,Y 576.129,Z 240.97,A -85,B 0,C 180,E1 27575.305,E2 27575.305} C_VEL
LIN {X 0,Y 576.082,Z 240.972,A -85,B 0,C 180,E1 27572.114,E2 27572.114} C_VEL
LIN {X 0,Y 576.145,Z 240.971,A -85,B 0,C 180,E1 27569.074,E2 27569.074} C_VEL
LIN {X 0,Y 576.076,Z 240.972,A -85,B 0,C 180,E1 27565.938,E2 27565.938} C_VEL
LIN {X 0,Y 576.145,Z 240.972,A -85,B 0,C 180,E1 27562.769,E2 27562.769} C_VEL
LIN {X 0,Y 576.074,Z 240.975,A -85,B 0,C 180,E1 27559.678,E2 27559.678} C_VEL
LIN {X 0,Y 576.157,Z 241.216,A -85,B 0,C 180,E1 27559.069,E2 27559.069} C_VEL
LIN {X 0,Y 577.527,Z 244.576,A -85,B 0,C 180,E1 27558.927,E2 27558.927} C_VEL
LIN {X 0,Y 580.918,Z 250.447,A -85,B 0,C 180,E1 27558.617,E2 27558.617} C_VEL
LIN {X 0,Y 580.009,Z 487.09,A -85,B 0,C 180,E1 27555.291,E2 27555.291} C_VEL
LIN {X 0,Y 579.796,Z 530.471,A -85,B 0,C 180,E1 27554.655,E2 27554.655} C_VEL
LIN {X 0,Y 579.573,Z 552.255,A -85,B 0,C 180,E1 27554.141,E2 27554.141} C_VEL
LIN {X 0,Y 579.203,Z 574.286,A -85,B 0,C 180,E1 27553.427,E2 27553.427} C_VEL
LIN {X 0,Y 578.883,Z 594.863,A -85,B 0,C 180,E1 27552.571,E2 27552.571} C_VEL
LIN {X 0,Y 578.485,Z 615.427,A -85,B 0,C 180,E1 27551.511,E2 27551.511} C_VEL
LIN {X 0,Y 578.051,Z 634.783,A -85,B 0,C 180,E1 27550.314,E2 27550.314} C_VEL
LIN {X 0,Y 577.658,Z 654.008,A -85,B 0,C 180,E1 27548.913,E2 27548.913} C_VEL
LIN {X 0,Y 577.274,Z 672.137,A -85,B 0,C 180,E1 27547.365,E2 27547.365} C_VEL
LIN {X 0,Y 576.921,Z 689.131,A -85,B 0,C 180,E1 27545.67,E2 27545.67} C_VEL
LIN {X 0,Y 576.617,Z 704.554,A -85,B 0,C 180,E1 27543.879,E2 27543.879} C_VEL
LIN {X 0,Y 576.386,Z 718.552,A -85,B 0,C 180,E1 27541.99,E2 27541.99} C_VEL
LIN {X 0,Y 576.21,Z 731.163,A -85,B 0,C 180,E1 27540.001,E2 27540.001} C_VEL
LIN {X 0,Y 576.083,Z 741.807,A -85,B 0,C 180,E1 27538.012,E2 27538.012} C_VEL
LIN {X 0,Y 575.994,Z 751.06,A -85,B 0,C 180,E1 27535.92,E2 27535.92} C_VEL
LIN {X 0,Y 575.951,Z 758.617,A -85,B 0,C 180,E1 27533.823,E2 27533.823} C_VEL
LIN {X 0,Y 575.927,Z 764.474,A -85,B 0,C 180,E1 27531.717,E2 27531.717} C_VEL
LIN {X 0,Y 575.908,Z 768.69,A -85,B 0,C 180,E1 27529.599,E2 27529.599} C_VEL
LIN {X 0,Y 575.904,Z 771.396,A -85,B 0,C 180,E1 27527.468,E2 27527.468} C_VEL
LIN {X 0,Y 575.915,Z 772.435,A -85,B 0,C 180,E1 27525.319,E2 27525.319} C_VEL
LIN {X 0,Y 575.913,Z 772.22,A -85,B 0,C 180,E1 27523.698,E2 27523.698} C_VEL
LIN {X 0,Y 574.912,Z 771.776,A -85,B 0,C 180,E1 27522.933,E2 27522.933} C_VEL
LIN {X 0,Y 568.567,Z 769.63,A -85,B 0,C 180,E1 27520.849,E2 27520.849} C_VEL
LIN {X 0,Y 567.918,Z 768.685,A -85,B 0,C 180,E1 27520.24,E2 27520.24} C_VEL
LIN {X 0,Y 567.928,Z 764.178,A -85,B 0,C 180,E1 27517.978,E2 27517.978} C_VEL
LIN {X 0,Y 567.965,Z 758.092,A -85,B 0,C 180,E1 27515.786,E2 27515.786} C_VEL
LIN {X 0,Y 568.028,Z 750.264,A -85,B 0,C 180,E1 27513.632,E2 27513.632} C_VEL
LIN {X 0,Y 568.139,Z 740.836,A -85,B 0,C 180,E1 27511.517,E2 27511.517} C_VEL
LIN {X 0,Y 568.319,Z 729.722,A -85,B 0,C 180,E1 27509.442,E2 27509.442} C_VEL
LIN {X 0,Y 568.56,Z 716.998,A -85,B 0,C 180,E1 27507.446,E2 27507.446} C_VEL
LIN {X 0,Y 568.861,Z 702.723,A -85,B 0,C 180,E1 27505.533,E2 27505.533} C_VEL
LIN {X 0,Y 569.247,Z 686.902,A -85,B 0,C 180,E1 27503.709,E2 27503.709} C_VEL
LIN {X 0,Y 569.707,Z 669.664,A -85,B 0,C 180,E1 27502.001,E2 27502.001} C_VEL
LIN {X 0,Y 570.212,Z 651.641,A -85,B 0,C 180,E1 27500.47,E2 27500.47} C_VEL
LIN {X 0,Y 570.741,Z 632.204,A -85,B 0,C 180,E1 27499.069,E2 27499.069} C_VEL
LIN {X 0,Y 571.251,Z 611.988,A -85,B 0,C 180,E1 27497.84,E2 27497.84} C_VEL
LIN {X 0,Y 571.777,Z 591.286,A -85,B 0,C 180,E1 27496.798,E2 27496.798} C_VEL
LIN {X 0,Y 572.234,Z 570.122,A -85,B 0,C 180,E1 27495.942,E2 27495.942} C_VEL
LIN {X 0,Y 572.577,Z 547.819,A -85,B 0,C 180,E1 27495.254,E2 27495.254} C_VEL
LIN {X 0,Y 572.899,Z 525.061,A -85,B 0,C 180,E1 27494.762,E2 27494.762} C_VEL
LIN {X 0,Y 574.058,Z 293.125,A -85,B 0,C 180,E1 27491.465,E2 27491.465} C_VEL
LIN {X 0,Y 574.094,Z 252.994,A -85,B 0,C 180,E1 27490.876,E2 27490.876} C_VEL
LIN {X 0,Y 569.665,Z 245.696,A -85,B 0,C 180,E1 27490.465,E2 27490.465} C_VEL
LIN {X 0,Y 568.254,Z 242.42,A -85,B 0,C 180,E1 27490.318,E2 27490.318} C_VEL
LIN {X 0,Y 568.183,Z 241.959,A -85,B 0,C 180,E1 27490.302,E2 27490.302} C_VEL
LIN {X 0,Y 568.212,Z 241.936,A -85,B 0,C 180,E1 27487,E2 27487} C_VEL
LIN {X 0,Y 568.21,Z 241.954,A -85,B 0,C 180,E1 27483.663,E2 27483.663} C_VEL
LIN {X 0,Y 568.178,Z 241.957,A -85,B 0,C 180,E1 27480.335,E2 27480.335} C_VEL
LIN {X 0,Y 568.221,Z 241.958,A -85,B 0,C 180,E1 27477.086,E2 27477.086} C_VEL
LIN {X 0,Y 568.183,Z 241.955,A -85,B 0,C 180,E1 27473.876,E2 27473.876} C_VEL
LIN {X 0,Y 568.19,Z 241.958,A -85,B 0,C 180,E1 27470.499,E2 27470.499} C_VEL
LIN {X 0,Y 568.215,Z 241.953,A -85,B 0,C 180,E1 27467.301,E2 27467.301} C_VEL
LIN {X 0,Y 568.172,Z 241.955,A -85,B 0,C 180,E1 27464.056,E2 27464.056} C_VEL
LIN {X 0,Y 568.221,Z 241.957,A -85,B 0,C 180,E1 27460.853,E2 27460.853} C_VEL
LIN {X 0,Y 568.172,Z 241.955,A -85,B 0,C 180,E1 27457.687,E2 27457.687} C_VEL
LIN {X 0,Y 568.189,Z 241.958,A -85,B 0,C 180,E1 27454.341,E2 27454.341} C_VEL
LIN {X 0,Y 568.209,Z 241.952,A -85,B 0,C 180,E1 27451.11,E2 27451.11} C_VEL
LIN {X 0,Y 568.168,Z 241.956,A -85,B 0,C 180,E1 27447.883,E2 27447.883} C_VEL
LIN {X 0,Y 568.222,Z 241.955,A -85,B 0,C 180,E1 27444.65,E2 27444.65} C_VEL
LIN {X 0,Y 568.167,Z 241.954,A -85,B 0,C 180,E1 27441.477,E2 27441.477} C_VEL
LIN {X 0,Y 568.184,Z 241.958,A -85,B 0,C 180,E1 27438.12,E2 27438.12} C_VEL
LIN {X 0,Y 568.189,Z 241.954,A -85,B 0,C 180,E1 27435.009,E2 27435.009} C_VEL
LIN {X 0,Y 568.166,Z 241.957,A -85,B 0,C 180,E1 27431.746,E2 27431.746} C_VEL
LIN {X 0,Y 568.223,Z 241.955,A -85,B 0,C 180,E1 27428.532,E2 27428.532} C_VEL
LIN {X 0,Y 568.158,Z 241.956,A -85,B 0,C 180,E1 27425.351,E2 27425.351} C_VEL
LIN {X 0,Y 568.199,Z 241.958,A -85,B 0,C 180,E1 27422.092,E2 27422.092} C_VEL
LIN {X 0,Y 568.162,Z 241.957,A -85,B 0,C 180,E1 27419.08,E2 27419.08} C_VEL
LIN {X 0,Y 568.17,Z 241.959,A -85,B 0,C 180,E1 27415.729,E2 27415.729} C_VEL
LIN {X 0,Y 568.182,Z 241.955,A -85,B 0,C 180,E1 27412.69,E2 27412.69} C_VEL
LIN {X 0,Y 568.159,Z 241.958,A -85,B 0,C 180,E1 27409.482,E2 27409.482} C_VEL
LIN {X 0,Y 568.205,Z 241.957,A -85,B 0,C 180,E1 27406.388,E2 27406.388} C_VEL
LIN {X 0,Y 568.149,Z 241.958,A -85,B 0,C 180,E1 27403.2,E2 27403.2} C_VEL
LIN {X 0,Y 568.22,Z 241.959,A -85,B 0,C 180,E1 27400.056,E2 27400.056} C_VEL
LIN {X 0,Y 568.147,Z 241.959,A -85,B 0,C 180,E1 27396.97,E2 27396.97} C_VEL
LIN {X 0,Y 568.201,Z 241.96,A -85,B 0,C 180,E1 27393.781,E2 27393.781} C_VEL
LIN {X 0,Y 568.15,Z 241.957,A -85,B 0,C 180,E1 27390.685,E2 27390.685} C_VEL
LIN {X 0,Y 568.156,Z 241.959,A -85,B 0,C 180,E1 27387.292,E2 27387.292} C_VEL
LIN {X 0,Y 568.17,Z 241.957,A -85,B 0,C 180,E1 27384.281,E2 27384.281} C_VEL
LIN {X 0,Y 568.143,Z 241.959,A -85,B 0,C 180,E1 27381.038,E2 27381.038} C_VEL
LIN {X 0,Y 568.2,Z 241.958,A -85,B 0,C 180,E1 27377.934,E2 27377.934} C_VEL
LIN {X 0,Y 568.137,Z 241.959,A -85,B 0,C 180,E1 27374.783,E2 27374.783} C_VEL
LIN {X 0,Y 568.211,Z 241.96,A -85,B 0,C 180,E1 27371.673,E2 27371.673} C_VEL
LIN {X 0,Y 568.135,Z 241.96,A -85,B 0,C 180,E1 27368.495,E2 27368.495} C_VEL
LIN {X 0,Y 568.184,Z 241.96,A -85,B 0,C 180,E1 27365.35,E2 27365.35} C_VEL
LIN {X 0,Y 568.137,Z 241.96,A -85,B 0,C 180,E1 27362.318,E2 27362.318} C_VEL
LIN {X 0,Y 568.156,Z 241.96,A -85,B 0,C 180,E1 27358.99,E2 27358.99} C_VEL
LIN {X 0,Y 568.149,Z 241.96,A -85,B 0,C 180,E1 27356.063,E2 27356.063} C_VEL
LIN {X 0,Y 568.145,Z 241.959,A -85,B 0,C 180,E1 27352.719,E2 27352.719} C_VEL
LIN {X 0,Y 568.172,Z 241.96,A -85,B 0,C 180,E1 27349.761,E2 27349.761} C_VEL
LIN {X 0,Y 568.145,Z 241.958,A -85,B 0,C 180,E1 27346.566,E2 27346.566} C_VEL
LIN {X 0,Y 568.189,Z 241.96,A -85,B 0,C 180,E1 27343.541,E2 27343.541} C_VEL
LIN {X 0,Y 568.145,Z 241.958,A -85,B 0,C 180,E1 27340.358,E2 27340.358} C_VEL
LIN {X 0,Y 568.219,Z 241.958,A -85,B 0,C 180,E1 27337.223,E2 27337.223} C_VEL
LIN {X 0,Y 568.145,Z 241.958,A -85,B 0,C 180,E1 27334.061,E2 27334.061} C_VEL
LIN {X 0,Y 568.195,Z 241.957,A -85,B 0,C 180,E1 27330.827,E2 27330.827} C_VEL
LIN {X 0,Y 568.155,Z 241.959,A -85,B 0,C 180,E1 27327.775,E2 27327.775} C_VEL
LIN {X 0,Y 568.162,Z 241.958,A -85,B 0,C 180,E1 27324.373,E2 27324.373} C_VEL
LIN {X 0,Y 568.185,Z 241.96,A -85,B 0,C 180,E1 27321.339,E2 27321.339} C_VEL
LIN {X 0,Y 568.155,Z 241.959,A -85,B 0,C 180,E1 27318.106,E2 27318.106} C_VEL
LIN {X 0,Y 568.218,Z 241.96,A -85,B 0,C 180,E1 27314.978,E2 27314.978} C_VEL
LIN {X 0,Y 568.155,Z 241.96,A -85,B 0,C 180,E1 27311.832,E2 27311.832} C_VEL
LIN {X 0,Y 568.184,Z 242.031,A -85,B 0,C 180,E1 27309.324,E2 27309.324} C_VEL
LIN {X 0,Y 569.567,Z 245.514,A -85,B 0,C 180,E1 27308.952,E2 27308.952} C_VEL
LIN {X 0,Y 573.768,Z 255.734,A -85,B 0,C 180,E1 27307.87,E2 27307.87} C_VEL
LIN {X 0,Y 572.965,Z 298.151,A -85,B 0,C 180,E1 27304.915,E2 27304.915} C_VEL
LIN {X 0,Y 573.008,Z 303.269,A -85,B 0,C 180,E1 27304.595,E2 27304.595} C_VEL
LIN {X 0,Y 574.382,Z 311.41,A -85,B 0,C 180,E1 27304.379,E2 27304.379} C_VEL
LIN {X 0,Y 573.264,Z 532.201,A -85,B 0,C 180,E1 27301.23,E2 27301.23} C_VEL
LIN {X 0,Y 572.869,Z 609.142,A -85,B 0,C 180,E1 27300.122,E2 27300.122} C_VEL
LIN {X 0,Y 572.544,Z 630.439,A -85,B 0,C 180,E1 27299.627,E2 27299.627} C_VEL
LIN {X 0,Y 572.143,Z 652.617,A -85,B 0,C 180,E1 27298.918,E2 27298.918} C_VEL
LIN {X 0,Y 571.744,Z 673.422,A -85,B 0,C 180,E1 27298.06,E2 27298.06} C_VEL
LIN {X 0,Y 571.221,Z 692.771,A -85,B 0,C 180,E1 27297.07,E2 27297.07} C_VEL
LIN {X 0,Y 570.705,Z 713.172,A -85,B 0,C 180,E1 27295.82,E2 27295.82} C_VEL
LIN {X 0,Y 570.2,Z 732.134,A -85,B 0,C 180,E1 27294.444,E2 27294.444} C_VEL
LIN {X 0,Y 569.698,Z 749.914,A -85,B 0,C 180,E1 27292.93,E2 27292.93} C_VEL
LIN {X 0,Y 569.254,Z 766.55,A -85,B 0,C 180,E1 27291.281,E2 27291.281} C_VEL
LIN {X 0,Y 568.877,Z 782.029,A -85,B 0,C 180,E1 27289.507,E2 27289.507} C_VEL
LIN {X 0,Y 568.581,Z 796.276,A -85,B 0,C 180,E1 27287.614,E2 27287.614} C_VEL
LIN {X 0,Y 568.331,Z 809.11,A -85,B 0,C 180,E1 27285.614,E2 27285.614} C_VEL
LIN {X 0,Y 568.148,Z 819.818,A -85,B 0,C 180,E1 27283.639,E2 27283.639} C_VEL
LIN {X 0,Y 568.036,Z 829.256,A -85,B 0,C 180,E1 27281.575,E2 27281.575} C_VEL
LIN {X 0,Y 567.965,Z 836.888,A -85,B 0,C 180,E1 27279.524,E2 27279.524} C_VEL
LIN {X 0,Y 567.928,Z 843.147,A -85,B 0,C 180,E1 27277.383,E2 27277.383} C_VEL
LIN {X 0,Y 567.921,Z 847.826,A -85,B 0,C 180,E1 27275.252,E2 27275.252} C_VEL
LIN {X 0,Y 567.916,Z 850.786,A -85,B 0,C 180,E1 27273.128,E2 27273.128} C_VEL
LIN {X 0,Y 567.91,Z 852.307,A -85,B 0,C 180,E1 27270.907,E2 27270.907} C_VEL
LIN {X 0,Y 567.91,Z 852.238,A -85,B 0,C 180,E1 27268.788,E2 27268.788} C_VEL
LIN {X 0,Y 567.914,Z 850.491,A -85,B 0,C 180,E1 27266.608,E2 27266.608} C_VEL
LIN {X 0,Y 567.921,Z 847.013,A -85,B 0,C 180,E1 27264.341,E2 27264.341} C_VEL
LIN {X 0,Y 567.941,Z 842.126,A -85,B 0,C 180,E1 27262.208,E2 27262.208} C_VEL
LIN {X 0,Y 567.97,Z 835.817,A -85,B 0,C 180,E1 27260.167,E2 27260.167} C_VEL
LIN {X 0,Y 568.048,Z 827.976,A -85,B 0,C 180,E1 27258.115,E2 27258.115} C_VEL
LIN {X 0,Y 568.159,Z 818.769,A -85,B 0,C 180,E1 27256.152,E2 27256.152} C_VEL
LIN {X 0,Y 568.348,Z 807.186,A -85,B 0,C 180,E1 27254.071,E2 27254.071} C_VEL
LIN {X 0,Y 568.608,Z 794.871,A -85,B 0,C 180,E1 27252.183,E2 27252.183} C_VEL
LIN {X 0,Y 568.928,Z 780.312,A -85,B 0,C 180,E1 27250.279,E2 27250.279} C_VEL
LIN {X 0,Y 569.299,Z 765.097,A -85,B 0,C 180,E1 27248.566,E2 27248.566} C_VEL
LIN {X 0,Y 569.759,Z 747.475,A -85,B 0,C 180,E1 27246.852,E2 27246.852} C_VEL
LIN {X 0,Y 570.245,Z 730.014,A -85,B 0,C 180,E1 27245.39,E2 27245.39} C_VEL
LIN {X 0,Y 570.753,Z 711.706,A -85,B 0,C 180,E1 27244.082,E2 27244.082} C_VEL
LIN {X 0,Y 571.25,Z 691.74,A -85,B 0,C 180,E1 27242.873,E2 27242.873} C_VEL
LIN {X 0,Y 571.761,Z 672.116,A -85,B 0,C 180,E1 27241.882,E2 27241.882} C_VEL
LIN {X 0,Y 572.171,Z 651.736,A -85,B 0,C 180,E1 27241.049,E2 27241.049} C_VEL
LIN {X 0,Y 572.553,Z 629.717,A -85,B 0,C 180,E1 27240.353,E2 27240.353} C_VEL
LIN {X 0,Y 572.878,Z 608.261,A -85,B 0,C 180,E1 27239.863,E2 27239.863} C_VEL
LIN {X 0,Y 573.633,Z 456.606,A -85,B 0,C 180,E1 27237.702,E2 27237.702} C_VEL
LIN {X 0,Y 574.223,Z 309.383,A -85,B 0,C 180,E1 27235.58,E2 27235.58} C_VEL
LIN {X 0,Y 572.879,Z 302.314,A -85,B 0,C 180,E1 27235.37,E2 27235.37} C_VEL
LIN {X 0,Y 573.632,Z 261.431,A -85,B 0,C 180,E1 27232.531,E2 27232.531} C_VEL
LIN {X 0,Y 573.591,Z 255.115,A -85,B 0,C 180,E1 27232.072,E2 27232.072} C_VEL
LIN {X 0,Y 568.21,Z 242.215,A -85,B 0,C 180,E1 27230.692,E2 27230.692} C_VEL
LIN {X 0,Y 568.183,Z 241.961,A -85,B 0,C 180,E1 27229.639,E2 27229.639} C_VEL
LIN {X 0,Y 568.154,Z 241.961,A -85,B 0,C 180,E1 27226.327,E2 27226.327} C_VEL
LIN {X 0,Y 568.218,Z 241.959,A -85,B 0,C 180,E1 27223.197,E2 27223.197} C_VEL
LIN {X 0,Y 568.147,Z 241.96,A -85,B 0,C 180,E1 27220.044,E2 27220.044} C_VEL
LIN {X 0,Y 568.205,Z 241.961,A -85,B 0,C 180,E1 27216.874,E2 27216.874} C_VEL
LIN {X 0,Y 568.148,Z 241.96,A -85,B 0,C 180,E1 27213.788,E2 27213.788} C_VEL
LIN {X 0,Y 568.162,Z 241.961,A -85,B 0,C 180,E1 27210.453,E2 27210.453} C_VEL
LIN {X 0,Y 568.158,Z 241.961,A -85,B 0,C 180,E1 27207.457,E2 27207.457} C_VEL
LIN {X 0,Y 568.145,Z 241.962,A -85,B 0,C 180,E1 27204.209,E2 27204.209} C_VEL
LIN {X 0,Y 568.165,Z 241.963,A -85,B 0,C 180,E1 27201.256,E2 27201.256} C_VEL
LIN {X 0,Y 568.149,Z 242.044,A -85,B 0,C 180,E1 27199.605,E2 27199.605} C_VEL
LIN {X 0,Y 569.465,Z 245.469,A -85,B 0,C 180,E1 27199.462,E2 27199.462} C_VEL
LIN {X 0,Y 571.169,Z 248.09,A -85,B 0,C 180,E1 27199.306,E2 27199.306} C_VEL
LIN {X 0,Y 574.245,Z 253.689,A -85,B 0,C 180,E1 27199.013,E2 27199.013} C_VEL
LIN {X 0,Y 573.091,Z 489.867,A -85,B 0,C 180,E1 27195.656,E2 27195.656} C_VEL
LIN {X 0,Y 572.834,Z 530.811,A -85,B 0,C 180,E1 27195.046,E2 27195.046} C_VEL
LIN {X 0,Y 572.544,Z 552.893,A -85,B 0,C 180,E1 27194.517,E2 27194.517} C_VEL
LIN {X 0,Y 572.093,Z 574.573,A -85,B 0,C 180,E1 27193.803,E2 27193.803} C_VEL
LIN {X 0,Y 571.649,Z 596.136,A -85,B 0,C 180,E1 27192.887,E2 27192.887} C_VEL
LIN {X 0,Y 571.16,Z 616.451,A -85,B 0,C 180,E1 27191.82,E2 27191.82} C_VEL
LIN {X 0,Y 570.611,Z 636.165,A -85,B 0,C 180,E1 27190.573,E2 27190.573} C_VEL
LIN {X 0,Y 570.099,Z 655.419,A -85,B 0,C 180,E1 27189.134,E2 27189.134} C_VEL
LIN {X 0,Y 569.621,Z 673.362,A -85,B 0,C 180,E1 27187.566,E2 27187.566} C_VEL
LIN {X 0,Y 569.179,Z 690.194,A -85,B 0,C 180,E1 27185.849,E2 27185.849} C_VEL
LIN {X 0,Y 568.803,Z 705.477,A -85,B 0,C 180,E1 27184.033,E2 27184.033} C_VEL
LIN {X 0,Y 568.509,Z 719.327,A -85,B 0,C 180,E1 27182.118,E2 27182.118} C_VEL
LIN {X 0,Y 568.284,Z 731.798,A -85,B 0,C 180,E1 27180.102,E2 27180.102} C_VEL
LIN {X 0,Y 568.128,Z 742.368,A -85,B 0,C 180,E1 27178.085,E2 27178.085} C_VEL
LIN {X 0,Y 568.016,Z 751.508,A -85,B 0,C 180,E1 27175.964,E2 27175.964} C_VEL
LIN {X 0,Y 567.955,Z 759.253,A -85,B 0,C 180,E1 27173.735,E2 27173.735} C_VEL
LIN {X 0,Y 567.933,Z 764.987,A -85,B 0,C 180,E1 27171.599,E2 27171.599} C_VEL
LIN {X 0,Y 567.916,Z 769.027,A -85,B 0,C 180,E1 27169.451,E2 27169.451} C_VEL
LIN {X 0,Y 567.913,Z 771.62,A -85,B 0,C 180,E1 27167.185,E2 27167.185} C_VEL
LIN {X 0,Y 567.917,Z 772.496,A -85,B 0,C 180,E1 27165.003,E2 27165.003} C_VEL
LIN {X 0,Y 567.913,Z 771.669,A -85,B 0,C 180,E1 27162.798,E2 27162.798} C_VEL
LIN {X 0,Y 567.915,Z 769.196,A -85,B 0,C 180,E1 27160.566,E2 27160.566} C_VEL
LIN {X 0,Y 567.918,Z 768.685,A -85,B 0,C 180,E1 27160.24,E2 27160.24} C_VEL
LIN {X 0,Y 566.916,Z 767.42,A -85,B 0,C 180,E1 27159.473,E2 27159.473} C_VEL
LIN {X 0,Y 560.588,Z 763.042,A -85,B 0,C 180,E1 27157.394,E2 27157.394} C_VEL
LIN {X 0,Y 559.944,Z 761.437,A -85,B 0,C 180,E1 27156.792,E2 27156.792} C_VEL
LIN {X 0,Y 560.006,Z 754.583,A -85,B 0,C 180,E1 27154.614,E2 27154.614} C_VEL
LIN {X 0,Y 560.112,Z 746.081,A -85,B 0,C 180,E1 27152.464,E2 27152.464} C_VEL
LIN {X 0,Y 560.286,Z 735.97,A -85,B 0,C 180,E1 27150.352,E2 27150.352} C_VEL
LIN {X 0,Y 560.54,Z 723.915,A -85,B 0,C 180,E1 27148.253,E2 27148.253} C_VEL
LIN {X 0,Y 560.888,Z 710.387,A -85,B 0,C 180,E1 27146.257,E2 27146.257} C_VEL
LIN {X 0,Y 561.319,Z 695.031,A -85,B 0,C 180,E1 27144.318,E2 27144.318} C_VEL
LIN {X 0,Y 561.832,Z 678.583,A -85,B 0,C 180,E1 27142.535,E2 27142.535} C_VEL
LIN {X 0,Y 562.418,Z 660.689,A -85,B 0,C 180,E1 27140.871,E2 27140.871} C_VEL
LIN {X 0,Y 563.051,Z 642.132,A -85,B 0,C 180,E1 27139.399,E2 27139.399} C_VEL
LIN {X 0,Y 563.673,Z 622.853,A -85,B 0,C 180,E1 27138.102,E2 27138.102} C_VEL
LIN {X 0,Y 564.297,Z 601.863,A -85,B 0,C 180,E1 27136.92,E2 27136.92} C_VEL
LIN {X 0,Y 564.927,Z 580.381,A -85,B 0,C 180,E1 27135.938,E2 27135.938} C_VEL
LIN {X 0,Y 565.421,Z 558.375,A -85,B 0,C 180,E1 27135.153,E2 27135.153} C_VEL
LIN {X 0,Y 565.793,Z 536.792,A -85,B 0,C 180,E1 27134.584,E2 27134.584} C_VEL
LIN {X 0,Y 566.083,Z 513.812,A -85,B 0,C 180,E1 27134.178,E2 27134.178} C_VEL
LIN {X 0,Y 567.429,Z 285.923,A -85,B 0,C 180,E1 27130.914,E2 27130.914} C_VEL
LIN {X 0,Y 567.407,Z 255.804,A -85,B 0,C 180,E1 27130.46,E2 27130.46} C_VEL
LIN {X 0,Y 561.707,Z 246.632,A -85,B 0,C 180,E1 27129.92,E2 27129.92} C_VEL
LIN {X 0,Y 560.306,Z 243.189,A -85,B 0,C 180,E1 27129.766,E2 27129.766} C_VEL
LIN {X 0,Y 560.246,Z 242.929,A -85,B 0,C 180,E1 27126.577,E2 27126.577} C_VEL
LIN {X 0,Y 560.282,Z 242.945,A -85,B 0,C 180,E1 27123.343,E2 27123.343} C_VEL
LIN {X 0,Y 560.243,Z 242.945,A -85,B 0,C 180,E1 27120.057,E2 27120.057} C_VEL
LIN {X 0,Y 560.263,Z 242.949,A -85,B 0,C 180,E1 27116.727,E2 27116.727} C_VEL
LIN {X 0,Y 560.274,Z 242.942,A -85,B 0,C 180,E1 27113.452,E2 27113.452} C_VEL
LIN {X 0,Y 560.237,Z 242.946,A -85,B 0,C 180,E1 27110.149,E2 27110.149} C_VEL
LIN {X 0,Y 560.283,Z 242.947,A -85,B 0,C 180,E1 27106.912,E2 27106.912} C_VEL
LIN {X 0,Y 560.245,Z 242.942,A -85,B 0,C 180,E1 27103.627,E2 27103.627} C_VEL
LIN {X 0,Y 560.242,Z 242.947,A -85,B 0,C 180,E1 27100.281,E2 27100.281} C_VEL
LIN {X 0,Y 560.286,Z 242.941,A -85,B 0,C 180,E1 27097.074,E2 27097.074} C_VEL
LIN {X 0,Y 560.23,Z 242.944,A -85,B 0,C 180,E1 27093.787,E2 27093.787} C_VEL
LIN {X 0,Y 560.273,Z 242.947,A -85,B 0,C 180,E1 27090.512,E2 27090.512} C_VEL
LIN {X 0,Y 560.242,Z 242.943,A -85,B 0,C 180,E1 27087.341,E2 27087.341} C_VEL
LIN {X 0,Y 560.232,Z 242.946,A -85,B 0,C 180,E1 27083.957,E2 27083.957} C_VEL
LIN {X 0,Y 560.284,Z 242.941,A -85,B 0,C 180,E1 27080.759,E2 27080.759} C_VEL
LIN {X 0,Y 560.226,Z 242.944,A -85,B 0,C 180,E1 27077.476,E2 27077.476} C_VEL
LIN {X 0,Y 560.253,Z 242.947,A -85,B 0,C 180,E1 27074.155,E2 27074.155} C_VEL
LIN {X 0,Y 560.241,Z 242.944,A -85,B 0,C 180,E1 27071.047,E2 27071.047} C_VEL
LIN {X 0,Y 560.228,Z 242.947,A -85,B 0,C 180,E1 27067.769,E2 27067.769} C_VEL
LIN {X 0,Y 560.271,Z 242.943,A -85,B 0,C 180,E1 27064.642,E2 27064.642} C_VEL
LIN {X 0,Y 560.219,Z 242.945,A -85,B 0,C 180,E1 27061.409,E2 27061.409} C_VEL
LIN {X 0,Y 560.277,Z 242.947,A -85,B 0,C 180,E1 27058.236,E2 27058.236} C_VEL
LIN {X 0,Y 560.221,Z 242.947,A -85,B 0,C 180,E1 27055.049,E2 27055.049} C_VEL
LIN {X 0,Y 560.237,Z 242.949,A -85,B 0,C 180,E1 27051.737,E2 27051.737} C_VEL
LIN {X 0,Y 560.238,Z 242.945,A -85,B 0,C 180,E1 27048.676,E2 27048.676} C_VEL
LIN {X 0,Y 560.217,Z 242.948,A -85,B 0,C 180,E1 27045.405,E2 27045.405} C_VEL
LIN {X 0,Y 560.275,Z 242.946,A -85,B 0,C 180,E1 27042.22,E2 27042.22} C_VEL
LIN {X 0,Y 560.208,Z 242.946,A -85,B 0,C 180,E1 27039.05,E2 27039.05} C_VEL
LIN {X 0,Y 560.264,Z 242.947,A -85,B 0,C 180,E1 27035.825,E2 27035.825} C_VEL
LIN {X 0,Y 560.211,Z 242.948,A -85,B 0,C 180,E1 27032.735,E2 27032.735} C_VEL
LIN {X 0,Y 560.224,Z 242.948,A -85,B 0,C 180,E1 27029.391,E2 27029.391} C_VEL
LIN {X 0,Y 560.227,Z 242.947,A -85,B 0,C 180,E1 27026.375,E2 27026.375} C_VEL
LIN {X 0,Y 560.209,Z 242.948,A -85,B 0,C 180,E1 27023.118,E2 27023.118} C_VEL
LIN {X 0,Y 560.251,Z 242.947,A -85,B 0,C 180,E1 27020.037,E2 27020.037} C_VEL
LIN {X 0,Y 560.2,Z 242.948,A -85,B 0,C 180,E1 27016.805,E2 27016.805} C_VEL
LIN {X 0,Y 560.268,Z 242.949,A -85,B 0,C 180,E1 27013.623,E2 27013.623} C_VEL
LIN {X 0,Y 560.2,Z 242.947,A -85,B 0,C 180,E1 27010.452,E2 27010.452} C_VEL
LIN {X 0,Y 560.217,Z 242.948,A -85,B 0,C 180,E1 27007.115,E2 27007.115} C_VEL
LIN {X 0,Y 560.213,Z 242.949,A -85,B 0,C 180,E1 27004.092,E2 27004.092} C_VEL
LIN {X 0,Y 560.202,Z 242.947,A -85,B 0,C 180,E1 27000.817,E2 27000.817} C_VEL
LIN {X 0,Y 560.232,Z 242.949,A -85,B 0,C 180,E1 26997.851,E2 26997.851} C_VEL
LIN {X 0,Y 560.199,Z 242.947,A -85,B 0,C 180,E1 26994.571,E2 26994.571} C_VEL
LIN {X 0,Y 560.27,Z 242.948,A -85,B 0,C 180,E1 26991.481,E2 26991.481} C_VEL
LIN {X 0,Y 560.201,Z 242.948,A -85,B 0,C 180,E1 26988.259,E2 26988.259} C_VEL
LIN {X 0,Y 560.26,Z 242.947,A -85,B 0,C 180,E1 26985.108,E2 26985.108} C_VEL
LIN {X 0,Y 560.208,Z 242.948,A -85,B 0,C 180,E1 26982.014,E2 26982.014} C_VEL
LIN {X 0,Y 560.221,Z 242.947,A -85,B 0,C 180,E1 26978.647,E2 26978.647} C_VEL
LIN {X 0,Y 560.23,Z 242.948,A -85,B 0,C 180,E1 26975.651,E2 26975.651} C_VEL
LIN {X 0,Y 560.213,Z 242.947,A -85,B 0,C 180,E1 26972.351,E2 26972.351} C_VEL
LIN {X 0,Y 560.275,Z 242.949,A -85,B 0,C 180,E1 26969.19,E2 26969.19} C_VEL
LIN {X 0,Y 560.21,Z 242.948,A -85,B 0,C 180,E1 26966.038,E2 26966.038} C_VEL
LIN {X 0,Y 560.28,Z 242.946,A -85,B 0,C 180,E1 26962.901,E2 26962.901} C_VEL
LIN {X 0,Y 560.216,Z 242.949,A -85,B 0,C 180,E1 26959.752,E2 26959.752} C_VEL
LIN {X 0,Y 560.241,Z 242.949,A -85,B 0,C 180,E1 26956.432,E2 26956.432} C_VEL
LIN {X 0,Y 560.233,Z 242.951,A -85,B 0,C 180,E1 26953.4,E2 26953.4} C_VEL
LIN {X 0,Y 560.221,Z 242.944,A -85,B 0,C 180,E1 26950.034,E2 26950.034} C_VEL
LIN {X 0,Y 560.245,Z 243.145,A -85,B 0,C 180,E1 26949.907,E2 26949.907} C_VEL
LIN {X 0,Y 561.505,Z 246.398,A -85,B 0,C 180,E1 26949.553,E2 26949.553} C_VEL
LIN {X 0,Y 566.972,Z 259.367,A -85,B 0,C 180,E1 26948.138,E2 26948.138} C_VEL
LIN {X 0,Y 566.021,Z 300.771,A -85,B 0,C 180,E1 26945.221,E2 26945.221} C_VEL
LIN {X 0,Y 566.122,Z 303.343,A -85,B 0,C 180,E1 26945.076,E2 26945.076} C_VEL
LIN {X 0,Y 567.768,Z 312.909,A -85,B 0,C 180,E1 26944.815,E2 26944.815} C_VEL
LIN {X 0,Y 566.416,Z 533.346,A -85,B 0,C 180,E1 26941.635,E2 26941.635} C_VEL
LIN {X 0,Y 565.942,Z 609.244,A -85,B 0,C 180,E1 26940.528,E2 26940.528} C_VEL
LIN {X 0,Y 565.548,Z 630.699,A -85,B 0,C 180,E1 26940.024,E2 26940.024} C_VEL
LIN {X 0,Y 565.085,Z 652.527,A -85,B 0,C 180,E1 26939.318,E2 26939.318} C_VEL
LIN {X 0,Y 564.579,Z 673.421,A -85,B 0,C 180,E1 26938.449,E2 26938.449} C_VEL
LIN {X 0,Y 563.935,Z 693.769,A -85,B 0,C 180,E1 26937.392,E2 26937.392} C_VEL
LIN {X 0,Y 563.301,Z 714.163,A -85,B 0,C 180,E1 26936.115,E2 26936.115} C_VEL
LIN {X 0,Y 562.7,Z 732.387,A -85,B 0,C 180,E1 26934.77,E2 26934.77} C_VEL
LIN {X 0,Y 562.101,Z 750.241,A -85,B 0,C 180,E1 26933.228,E2 26933.228} C_VEL
LIN {X 0,Y 561.571,Z 766.699,A -85,B 0,C 180,E1 26931.57,E2 26931.57} C_VEL
LIN {X 0,Y 561.083,Z 782.88,A -85,B 0,C 180,E1 26929.681,E2 26929.681} C_VEL
LIN {X 0,Y 560.714,Z 797.05,A -85,B 0,C 180,E1 26927.752,E2 26927.752} C_VEL
LIN {X 0,Y 560.417,Z 809.744,A -85,B 0,C 180,E1 26925.734,E2 26925.734} C_VEL
LIN {X 0,Y 560.198,Z 820.338,A -85,B 0,C 180,E1 26923.731,E2 26923.731} C_VEL
LIN {X 0,Y 560.057,Z 830.072,A -85,B 0,C 180,E1 26921.533,E2 26921.533} C_VEL
LIN {X 0,Y 559.982,Z 837.939,A -85,B 0,C 180,E1 26919.35,E2 26919.35} C_VEL
LIN {X 0,Y 559.938,Z 843.91,A -85,B 0,C 180,E1 26917.179,E2 26917.179} C_VEL
LIN {X 0,Y 559.917,Z 848.582,A -85,B 0,C 180,E1 26914.841,E2 26914.841} C_VEL
LIN {X 0,Y 559.906,Z 851.339,A -85,B 0,C 180,E1 26912.66,E2 26912.66} C_VEL
LIN {X 0,Y 559.898,Z 852.395,A -85,B 0,C 180,E1 26910.511,E2 26910.511} C_VEL
LIN {X 0,Y 559.901,Z 851.948,A -85,B 0,C 180,E1 26908.259,E2 26908.259} C_VEL
LIN {X 0,Y 559.909,Z 849.993,A -85,B 0,C 180,E1 26906.108,E2 26906.108} C_VEL
LIN {X 0,Y 559.922,Z 846.395,A -85,B 0,C 180,E1 26903.951,E2 26903.951} C_VEL
LIN {X 0,Y 559.958,Z 841.278,A -85,B 0,C 180,E1 26901.786,E2 26901.786} C_VEL
LIN {X 0,Y 560.011,Z 834.753,A -85,B 0,C 180,E1 26899.714,E2 26899.714} C_VEL
LIN {X 0,Y 560.11,Z 826.136,A -85,B 0,C 180,E1 26897.525,E2 26897.525} C_VEL
LIN {X 0,Y 560.287,Z 816.115,A -85,B 0,C 180,E1 26895.426,E2 26895.426} C_VEL
LIN {X 0,Y 560.526,Z 804.622,A -85,B 0,C 180,E1 26893.416,E2 26893.416} C_VEL
LIN {X 0,Y 560.837,Z 791.783,A -85,B 0,C 180,E1 26891.497,E2 26891.497} C_VEL
LIN {X 0,Y 561.234,Z 777.65,A -85,B 0,C 180,E1 26889.671,E2 26889.671} C_VEL
LIN {X 0,Y 561.729,Z 761.822,A -85,B 0,C 180,E1 26887.907,E2 26887.907} C_VEL
LIN {X 0,Y 562.275,Z 745.058,A -85,B 0,C 180,E1 26886.303,E2 26886.303} C_VEL
LIN {X 0,Y 562.893,Z 726.382,A -85,B 0,C 180,E1 26884.766,E2 26884.766} C_VEL
LIN {X 0,Y 563.512,Z 707.519,A -85,B 0,C 180,E1 26883.439,E2 26883.439} C_VEL
LIN {X 0,Y 564.134,Z 687.734,A -85,B 0,C 180,E1 26882.273,E2 26882.273} C_VEL
LIN {X 0,Y 564.708,Z 667.027,A -85,B 0,C 180,E1 26881.267,E2 26881.267} C_VEL
LIN {X 0,Y 565.265,Z 645.645,A -85,B 0,C 180,E1 26880.436,E2 26880.436} C_VEL
LIN {X 0,Y 565.672,Z 624.866,A -85,B 0,C 180,E1 26879.819,E2 26879.819} C_VEL
LIN {X 0,Y 565.99,Z 603.245,A -85,B 0,C 180,E1 26879.372,E2 26879.372} C_VEL
LIN {X 0,Y 567.329,Z 377.375,A -85,B 0,C 180,E1 26876.123,E2 26876.123} C_VEL
LIN {X 0,Y 567.592,Z 310.839,A -85,B 0,C 180,E1 26875.142,E2 26875.142} C_VEL
LIN {X 0,Y 565.985,Z 302.201,A -85,B 0,C 180,E1 26874.878,E2 26874.878} C_VEL
LIN {X 0,Y 566.913,Z 261.431,A -85,B 0,C 180,E1 26872.009,E2 26872.009} C_VEL
LIN {X 0,Y 566.817,Z 258.695,A -85,B 0,C 180,E1 26871.8,E2 26871.8} C_VEL
LIN {X 0,Y 561.503,Z 246.401,A -85,B 0,C 180,E1 26870.447,E2 26870.447} C_VEL
LIN {X 0,Y 560.218,Z 242.952,A -85,B 0,C 180,E1 26870.07,E2 26870.07} C_VEL
LIN {X 0,Y 560.256,Z 242.95,A -85,B 0,C 180,E1 26866.88,E2 26866.88} C_VEL
LIN {X 0,Y 560.219,Z 242.949,A -85,B 0,C 180,E1 26863.828,E2 26863.828} C_VEL
LIN {X 0,Y 560.216,Z 242.95,A -85,B 0,C 180,E1 26860.382,E2 26860.382} C_VEL
LIN {X 0,Y 560.25,Z 242.948,A -85,B 0,C 180,E1 26857.358,E2 26857.358} C_VEL
LIN {X 0,Y 560.206,Z 242.95,A -85,B 0,C 180,E1 26854.09,E2 26854.09} C_VEL
LIN {X 0,Y 560.271,Z 242.949,A -85,B 0,C 180,E1 26850.863,E2 26850.863} C_VEL
LIN {X 0,Y 560.205,Z 242.95,A -85,B 0,C 180,E1 26847.715,E2 26847.715} C_VEL
LIN {X 0,Y 560.216,Z 242.951,A -85,B 0,C 180,E1 26844.349,E2 26844.349} C_VEL
LIN {X 0,Y 560.217,Z 242.953,A -85,B 0,C 180,E1 26841.353,E2 26841.353} C_VEL
LIN {X 0,Y 560.235,Z 243.173,A -85,B 0,C 180,E1 26840.149,E2 26840.149} C_VEL
LIN {X 0,Y 561.554,Z 246.511,A -85,B 0,C 180,E1 26840.003,E2 26840.003} C_VEL
LIN {X 0,Y 563.468,Z 249.575,A -85,B 0,C 180,E1 26839.82,E2 26839.82} C_VEL
LIN {X 0,Y 567.602,Z 256.503,A -85,B 0,C 180,E1 26839.426,E2 26839.426} C_VEL
LIN {X 0,Y 566.199,Z 492.528,A -85,B 0,C 180,E1 26836.033,E2 26836.033} C_VEL
LIN {X 0,Y 565.897,Z 531.257,A -85,B 0,C 180,E1 26835.445,E2 26835.445} C_VEL
LIN {X 0,Y 565.536,Z 553.447,A -85,B 0,C 180,E1 26834.904,E2 26834.904} C_VEL
LIN {X 0,Y 565.014,Z 574.855,A -85,B 0,C 180,E1 26834.188,E2 26834.188} C_VEL
LIN {X 0,Y 564.473,Z 596.37,A -85,B 0,C 180,E1 26833.262,E2 26833.262} C_VEL
LIN {X 0,Y 563.868,Z 616.672,A -85,B 0,C 180,E1 26832.183,E2 26832.183} C_VEL
LIN {X 0,Y 563.24,Z 635.922,A -85,B 0,C 180,E1 26830.951,E2 26830.951} C_VEL
LIN {X 0,Y 562.599,Z 655.445,A -85,B 0,C 180,E1 26829.475,E2 26829.475} C_VEL
LIN {X 0,Y 562.003,Z 673.515,A -85,B 0,C 180,E1 26827.875,E2 26827.875} C_VEL
LIN {X 0,Y 561.462,Z 690.324,A -85,B 0,C 180,E1 26826.135,E2 26826.135} C_VEL
LIN {X 0,Y 561.013,Z 705.591,A -85,B 0,C 180,E1 26824.294,E2 26824.294} C_VEL
LIN {X 0,Y 560.65,Z 719.423,A -85,B 0,C 180,E1 26822.352,E2 26822.352} C_VEL
LIN {X 0,Y 560.373,Z 731.874,A -85,B 0,C 180,E1 26820.308,E2 26820.308} C_VEL
LIN {X 0,Y 560.178,Z 742.423,A -85,B 0,C 180,E1 26818.263,E2 26818.263} C_VEL
LIN {X 0,Y 560.042,Z 751.554,A -85,B 0,C 180,E1 26816.111,E2 26816.111} C_VEL
LIN {X 0,Y 559.967,Z 759.285,A -85,B 0,C 180,E1 26813.851,E2 26813.851} C_VEL
LIN {X 0,Y 559.934,Z 765.008,A -85,B 0,C 180,E1 26811.685,E2 26811.685} C_VEL
LIN {X 0,Y 559.914,Z 769.043,A -85,B 0,C 180,E1 26809.507,E2 26809.507} C_VEL
LIN {X 0,Y 559.913,Z 771.656,A -85,B 0,C 180,E1 26807.166,E2 26807.166} C_VEL
LIN {X 0,Y 559.917,Z 772.497,A -85,B 0,C 180,E1 26804.995,E2 26804.995} C_VEL
LIN {X 0,Y 559.912,Z 771.666,A -85,B 0,C 180,E1 26802.758,E2 26802.758} C_VEL
LIN {X 0,Y 559.916,Z 769.186,A -85,B 0,C 180,E1 26800.494,E2 26800.494} C_VEL
LIN {X 0,Y 559.93,Z 765.203,A -85,B 0,C 180,E1 26798.309,E2 26798.309} C_VEL
LIN {X 0,Y 559.944,Z 761.437,A -85,B 0,C 180,E1 26796.792,E2 26796.792} C_VEL
LIN {X 0,Y 558.949,Z 759.278,A -85,B 0,C 180,E1 26796.035,E2 26796.035} C_VEL
LIN {X 0,Y 552.797,Z 753.044,A -85,B 0,C 180,E1 26794.037,E2 26794.037} C_VEL
LIN {X 0,Y 552.082,Z 750.625,A -85,B 0,C 180,E1 26793.393,E2 26793.393} C_VEL
LIN {X 0,Y 552.248,Z 741.211,A -85,B 0,C 180,E1 26791.199,E2 26791.199} C_VEL
LIN {X 0,Y 552.498,Z 730.198,A -85,B 0,C 180,E1 26789.071,E2 26789.071} C_VEL
LIN {X 0,Y 552.851,Z 717.581,A -85,B 0,C 180,E1 26787.021,E2 26787.021} C_VEL
LIN {X 0,Y 553.309,Z 703.422,A -85,B 0,C 180,E1 26785.054,E2 26785.054} C_VEL
LIN {X 0,Y 553.873,Z 687.742,A -85,B 0,C 180,E1 26783.181,E2 26783.181} C_VEL
LIN {X 0,Y 554.533,Z 670.398,A -85,B 0,C 180,E1 26781.404,E2 26781.404} C_VEL
LIN {X 0,Y 555.221,Z 652.804,A -85,B 0,C 180,E1 26779.86,E2 26779.86} C_VEL
LIN {X 0,Y 555.976,Z 633.609,A -85,B 0,C 180,E1 26778.428,E2 26778.428} C_VEL
LIN {X 0,Y 556.714,Z 613.791,A -85,B 0,C 180,E1 26777.176,E2 26777.176} C_VEL
LIN {X 0,Y 557.432,Z 593.541,A -85,B 0,C 180,E1 26776.115,E2 26776.115} C_VEL
LIN {X 0,Y 558.089,Z 571.984,A -85,B 0,C 180,E1 26775.208,E2 26775.208} C_VEL
LIN {X 0,Y 558.613,Z 549.594,A -85,B 0,C 180,E1 26774.483,E2 26774.483} C_VEL
LIN {X 0,Y 559.075,Z 526.834,A -85,B 0,C 180,E1 26773.965,E2 26773.965} C_VEL
LIN {X 0,Y 560.72,Z 296.976,A -85,B 0,C 180,E1 26770.617,E2 26770.617} C_VEL
LIN {X 0,Y 560.811,Z 259.094,A -85,B 0,C 180,E1 26770.046,E2 26770.046} C_VEL
LIN {X 0,Y 553.98,Z 247.877,A -85,B 0,C 180,E1 26769.377,E2 26769.377} C_VEL
LIN {X 0,Y 552.46,Z 244.624,A -85,B 0,C 180,E1 26769.213,E2 26769.213} C_VEL
LIN {X 0,Y 552.343,Z 243.928,A -85,B 0,C 180,E1 26769.181,E2 26769.181} C_VEL
LIN {X 0,Y 552.325,Z 243.922,A -85,B 0,C 180,E1 26765.784,E2 26765.784} C_VEL
LIN {X 0,Y 552.304,Z 243.936,A -85,B 0,C 180,E1 26762.403,E2 26762.403} C_VEL
LIN {X 0,Y 552.344,Z 243.936,A -85,B 0,C 180,E1 26759.141,E2 26759.141} C_VEL
LIN {X 0,Y 552.308,Z 243.933,A -85,B 0,C 180,E1 26755.868,E2 26755.868} C_VEL
LIN {X 0,Y 552.308,Z 243.936,A -85,B 0,C 180,E1 26752.457,E2 26752.457} C_VEL
LIN {X 0,Y 552.343,Z 243.932,A -85,B 0,C 180,E1 26749.237,E2 26749.237} C_VEL
LIN {X 0,Y 552.296,Z 243.933,A -85,B 0,C 180,E1 26745.973,E2 26745.973} C_VEL
LIN {X 0,Y 552.334,Z 243.937,A -85,B 0,C 180,E1 26742.653,E2 26742.653} C_VEL
LIN {X 0,Y 552.32,Z 243.932,A -85,B 0,C 180,E1 26739.378,E2 26739.378} C_VEL
LIN {X 0,Y 552.294,Z 243.933,A -85,B 0,C 180,E1 26736.028,E2 26736.028} C_VEL
LIN {X 0,Y 552.344,Z 243.934,A -85,B 0,C 180,E1 26732.802,E2 26732.802} C_VEL
LIN {X 0,Y 552.293,Z 243.932,A -85,B 0,C 180,E1 26729.586,E2 26729.586} C_VEL
LIN {X 0,Y 552.303,Z 243.932,A -85,B 0,C 180,E1 26726.16,E2 26726.16} C_VEL
LIN {X 0,Y 552.339,Z 243.93,A -85,B 0,C 180,E1 26722.93,E2 26722.93} C_VEL
LIN {X 0,Y 552.287,Z 243.934,A -85,B 0,C 180,E1 26719.676,E2 26719.676} C_VEL
LIN {X 0,Y 552.339,Z 243.937,A -85,B 0,C 180,E1 26716.39,E2 26716.39} C_VEL
LIN {X 0,Y 552.297,Z 243.933,A -85,B 0,C 180,E1 26713.164,E2 26713.164} C_VEL
LIN {X 0,Y 552.288,Z 243.935,A -85,B 0,C 180,E1 26709.772,E2 26709.772} C_VEL
LIN {X 0,Y 552.344,Z 243.933,A -85,B 0,C 180,E1 26706.533,E2 26706.533} C_VEL
LIN {X 0,Y 552.281,Z 243.935,A -85,B 0,C 180,E1 26703.323,E2 26703.323} C_VEL
LIN {X 0,Y 552.316,Z 243.938,A -85,B 0,C 180,E1 26700.025,E2 26700.025} C_VEL
LIN {X 0,Y 552.297,Z 243.932,A -85,B 0,C 180,E1 26696.859,E2 26696.859} C_VEL
LIN {X 0,Y 552.28,Z 243.934,A -85,B 0,C 180,E1 26693.493,E2 26693.493} C_VEL
LIN {X 0,Y 552.344,Z 243.935,A -85,B 0,C 180,E1 26690.284,E2 26690.284} C_VEL
LIN {X 0,Y 552.274,Z 243.936,A -85,B 0,C 180,E1 26687.102,E2 26687.102} C_VEL
LIN {X 0,Y 552.32,Z 243.937,A -85,B 0,C 180,E1 26683.892,E2 26683.892} C_VEL
LIN {X 0,Y 552.279,Z 243.936,A -85,B 0,C 180,E1 26680.808,E2 26680.808} C_VEL
LIN {X 0,Y 552.278,Z 243.938,A -85,B 0,C 180,E1 26677.333,E2 26677.333} C_VEL
LIN {X 0,Y 552.33,Z 243.933,A -85,B 0,C 180,E1 26674.135,E2 26674.135} C_VEL
LIN {X 0,Y 552.267,Z 243.935,A -85,B 0,C 180,E1 26670.893,E2 26670.893} C_VEL
LIN {X 0,Y 552.322,Z 243.937,A -85,B 0,C 180,E1 26667.724,E2 26667.724} C_VEL
LIN {X 0,Y 552.269,Z 243.935,A -85,B 0,C 180,E1 26664.606,E2 26664.606} C_VEL
LIN {X 0,Y 552.275,Z 243.937,A -85,B 0,C 180,E1 26661.197,E2 26661.197} C_VEL
LIN {X 0,Y 552.298,Z 243.937,A -85,B 0,C 180,E1 26658.12,E2 26658.12} C_VEL
LIN {X 0,Y 552.262,Z 243.937,A -85,B 0,C 180,E1 26654.896,E2 26654.896} C_VEL
LIN {X 0,Y 552.33,Z 243.938,A -85,B 0,C 180,E1 26651.673,E2 26651.673} C_VEL
LIN {X 0,Y 552.26,Z 243.938,A -85,B 0,C 180,E1 26648.431,E2 26648.431} C_VEL
LIN {X 0,Y 552.277,Z 243.938,A -85,B 0,C 180,E1 26645.088,E2 26645.088} C_VEL
LIN {X 0,Y 552.275,Z 243.938,A -85,B 0,C 180,E1 26642.074,E2 26642.074} C_VEL
LIN {X 0,Y 552.263,Z 243.938,A -85,B 0,C 180,E1 26638.754,E2 26638.754} C_VEL
LIN {X 0,Y 552.315,Z 243.938,A -85,B 0,C 180,E1 26635.638,E2 26635.638} C_VEL
LIN {X 0,Y 552.26,Z 243.938,A -85,B 0,C 180,E1 26632.404,E2 26632.404} C_VEL
LIN {X 0,Y 552.327,Z 243.936,A -85,B 0,C 180,E1 26629.253,E2 26629.253} C_VEL
LIN {X 0,Y 552.269,Z 243.936,A -85,B 0,C 180,E1 26626.066,E2 26626.066} C_VEL
LIN {X 0,Y 552.283,Z 243.937,A -85,B 0,C 180,E1 26622.727,E2 26622.727} C_VEL
LIN {X 0,Y 552.293,Z 243.937,A -85,B 0,C 180,E1 26619.659,E2 26619.659} C_VEL
LIN {X 0,Y 552.27,Z 243.936,A -85,B 0,C 180,E1 26616.356,E2 26616.356} C_VEL
LIN {X 0,Y 552.339,Z 243.936,A -85,B 0,C 180,E1 26613.178,E2 26613.178} C_VEL
LIN {X 0,Y 552.269,Z 243.937,A -85,B 0,C 180,E1 26610.02,E2 26610.02} C_VEL
LIN {X 0,Y 552.314,Z 243.936,A -85,B 0,C 180,E1 26606.733,E2 26606.733} C_VEL
LIN {X 0,Y 552.282,Z 243.938,A -85,B 0,C 180,E1 26603.669,E2 26603.669} C_VEL
LIN {X 0,Y 552.284,Z 243.937,A -85,B 0,C 180,E1 26600.277,E2 26600.277} C_VEL
LIN {X 0,Y 552.327,Z 243.939,A -85,B 0,C 180,E1 26597.104,E2 26597.104} C_VEL
LIN {X 0,Y 552.278,Z 243.939,A -85,B 0,C 180,E1 26593.897,E2 26593.897} C_VEL
LIN {X 0,Y 552.341,Z 243.927,A -85,B 0,C 180,E1 26590.666,E2 26590.666} C_VEL
LIN {X 0,Y 552.328,Z 243.988,A -85,B 0,C 180,E1 26590.508,E2 26590.508} C_VEL
LIN {X 0,Y 553.735,Z 247.62,A -85,B 0,C 180,E1 26590.119,E2 26590.119} C_VEL
LIN {X 0,Y 560.173,Z 262.496,A -85,B 0,C 180,E1 26588.452,E2 26588.452} C_VEL
LIN {X 0,Y 559.129,Z 302.193,A -85,B 0,C 180,E1 26585.618,E2 26585.618} C_VEL
LIN {X 0,Y 561.189,Z 314.345,A -85,B 0,C 180,E1 26585.261,E2 26585.261} C_VEL
LIN {X 0,Y 559.592,Z 535,A -85,B 0,C 180,E1 26582.041,E2 26582.041} C_VEL
LIN {X 0,Y 559.046,Z 609.244,A -85,B 0,C 180,E1 26580.946,E2 26580.946} C_VEL
LIN {X 0,Y 558.583,Z 630.7,A -85,B 0,C 180,E1 26580.438,E2 26580.438} C_VEL
LIN {X 0,Y 558.05,Z 652.597,A -85,B 0,C 180,E1 26579.721,E2 26579.721} C_VEL
LIN {X 0,Y 557.44,Z 673.421,A -85,B 0,C 180,E1 26578.847,E2 26578.847} C_VEL
LIN {X 0,Y 556.703,Z 693.771,A -85,B 0,C 180,E1 26577.778,E2 26577.778} C_VEL
LIN {X 0,Y 555.95,Z 714.163,A -85,B 0,C 180,E1 26576.487,E2 26576.487} C_VEL
LIN {X 0,Y 555.2,Z 733.164,A -85,B 0,C 180,E1 26575.062,E2 26575.062} C_VEL
LIN {X 0,Y 554.505,Z 751.124,A -85,B 0,C 180,E1 26573.483,E2 26573.483} C_VEL
LIN {X 0,Y 553.868,Z 767.711,A -85,B 0,C 180,E1 26571.774,E2 26571.774} C_VEL
LIN {X 0,Y 553.322,Z 782.881,A -85,B 0,C 180,E1 26569.968,E2 26569.968} C_VEL
LIN {X 0,Y 552.872,Z 797.052,A -85,B 0,C 180,E1 26568.013,E2 26568.013} C_VEL
LIN {X 0,Y 552.515,Z 809.742,A -85,B 0,C 180,E1 26565.965,E2 26565.965} C_VEL
LIN {X 0,Y 552.258,Z 820.339,A -85,B 0,C 180,E1 26563.932,E2 26563.932} C_VEL
LIN {X 0,Y 552.085,Z 830.073,A -85,B 0,C 180,E1 26561.702,E2 26561.702} C_VEL
LIN {X 0,Y 551.99,Z 837.939,A -85,B 0,C 180,E1 26559.486,E2 26559.486} C_VEL
LIN {X 0,Y 551.939,Z 843.91,A -85,B 0,C 180,E1 26557.284,E2 26557.284} C_VEL
LIN {X 0,Y 551.919,Z 848.466,A -85,B 0,C 180,E1 26554.987,E2 26554.987} C_VEL
LIN {X 0,Y 551.909,Z 851.235,A -85,B 0,C 180,E1 26552.803,E2 26552.803} C_VEL
LIN {X 0,Y 551.898,Z 852.373,A -85,B 0,C 180,E1 26550.622,E2 26550.622} C_VEL
LIN {X 0,Y 551.899,Z 852.014,A -85,B 0,C 180,E1 26548.338,E2 26548.338} C_VEL
LIN {X 0,Y 551.905,Z 850.22,A -85,B 0,C 180,E1 26546.26,E2 26546.26} C_VEL
LIN {X 0,Y 551.923,Z 846.601,A -85,B 0,C 180,E1 26543.968,E2 26543.968} C_VEL
LIN {X 0,Y 551.965,Z 841.581,A -85,B 0,C 180,E1 26541.772,E2 26541.772} C_VEL
LIN {X 0,Y 552.026,Z 835.108,A -85,B 0,C 180,E1 26539.669,E2 26539.669} C_VEL
LIN {X 0,Y 552.146,Z 826.542,A -85,B 0,C 180,E1 26537.436,E2 26537.436} C_VEL
LIN {X 0,Y 552.351,Z 816.683,A -85,B 0,C 180,E1 26535.319,E2 26535.319} C_VEL
LIN {X 0,Y 552.633,Z 805.265,A -85,B 0,C 180,E1 26533.28,E2 26533.28} C_VEL
LIN {X 0,Y 553.028,Z 791.784,A -85,B 0,C 180,E1 26531.226,E2 26531.226} C_VEL
LIN {X 0,Y 553.514,Z 777.383,A -85,B 0,C 180,E1 26529.343,E2 26529.343} C_VEL
LIN {X 0,Y 554.098,Z 761.612,A -85,B 0,C 180,E1 26527.563,E2 26527.563} C_VEL
